// TIA Portal project "SimLogic" (V15)

(* hardware
DEVICE "S71500/ET200MP station_1"  S7-1500 station
   slot 0: "Rail_0"  Rack  6ES7 590-1***0-0AA0
   slot 1: "PLC_1"  CPU 1511-1 PN  6ES7 511-1AK00-0AB0  V1.8
      slot 3: "CPU display_1"  6ES7591-1AA00-0AA0
DEVICE "PC-System_1"  SIMATIC PC station
   slot 0: "SIMATIC PC station"  Rail  SIMATIC PC-Station  V1.0
      slot 125: "Stationmanager"  Station_Manager  V6.0.4
   slot 1: "HMI_RT_1"  WinCC RT Professional  6AV2 105-0xxxx-xxxx  15.0.0.0
   slot 2: "IE general_1"  IE General  IE_CP  V8.2.0
*)

// ===== PLC "PLC_1"  CPU 1511-1 PN =====

VAR_GLOBAL   // PLC tag table "Default tag table"
   "Brake_Out" AT %M0.0 : Bool;
   "Baffle_Out" AT %MW18 : Int;
   "RPM_In" AT %MW2 : Int;
   "OilTemp_In" AT %MW4 : Int;
   "Baffle_En" AT %M0.1 : Bool;
   "Current_In" AT %MW6 : Int;
   "OilPumpVFDsp_Out" AT %MW8 : Int;
   "OilPumpVFDen_Out" AT %M0.2 : Bool;
   "OilFlow_In" AT %MW10 : Int;
   "ProgLang" AT %MW12 : Int;
   "ONS1" AT %M0.3 : Bool;
   "PB_LAD" AT %M0.4 : Bool;
   "ONS" AT %M0.5 : Bool;
   "PB_FBD" AT %M0.6 : Bool;
   "PB_SCL" AT %M0.7 : Bool;
   "PB_STL" AT %M1.0 : Bool;
   "ONS2" AT %M1.1 : Bool;
   "ONS3" AT %M1.2 : Bool;
   "ONS4" AT %M1.3 : Bool;
   "AlarmHorn_Out" AT %M1.4 : Bool;
   "StationInterlock_Out" AT %M1.5 : Bool;
   "OilPumpVFDsp_Pct" AT %MW14 : Int;
   "Baffle_Pct" AT %MW16 : Int;
   "OilTemp" AT %MW20 : Int;
   "OilFlow" AT %MW22 : Int;
   "RPM" AT %MW24 : Int;
   "Current" AT %MW26 : Int;
   "OilPumpVFDOff_PB" AT %M1.6 : Bool;
   "OilPumpVFDHand_PB" AT %M1.7 : Bool;
   "OilPumpVFDAuto_PB" AT %M28.0 : Bool;
   "OilPumpVFD_HOA" AT %MW30 : Int;
   "Brake_HOA" AT %MW32 : Int;
   "BrakeOff_PB" AT %M28.1 : Bool;
   "BrakeHand_PB" AT %M28.2 : Bool;
   "BrakeAuto_PB" AT %M28.3 : Bool;
   "AlarmHorn_HOA" AT %MW34 : Int;
   "AlarmHornOff_PB" AT %M28.4 : Bool;
   "AlarmHornHand_PB" AT %M28.5 : Bool;
   "AlarmHornAuto_PB" AT %M28.6 : Bool;
   "StationIntOff_PB" AT %M28.7 : Bool;
   "StationIntHand_PB" AT %M29.0 : Bool;
   "StationIntAuto_PB" AT %M29.1 : Bool;
   "StationInt_HOA" AT %MW36 : Int;
   "StationInt" AT %M29.2 : Bool;
   "Brake_Ctrl" AT %M29.3 : Bool;
   "AlarmHorn_Ctrl" AT %M29.4 : Bool;
   "StationInt_Ctrl" AT %M29.5 : Bool;
   "OilPumpVFD_Ctrl" AT %M29.6 : Bool;
   "OilLowFlowDelay_SP" AT %MW38 : Int;
   "AlarmReset" AT %M29.7 : Bool;
   "AlarmSilence" AT %M40.0 : Bool;
   "OilLowFlowAlarm" AT %M40.1 : Bool;
   "OilLowFlowNotify" AT %M40.2 : Bool;
   "OilLowFlowAlarm_SP" AT %MW42 : Int;
   "OvercurrentDelay_SP" AT %MW44 : Int;
   "OvercurrentAlarm_SP" AT %MW46 : Int;
   "OvercurrentAlarm" AT %M40.3 : Bool;
   "OvercurrentNotify" AT %M40.4 : Bool;
   "HighOilTempDelay_SP" AT %MW48 : Int;
   "HighOilTempAlarm_SP" AT %MW50 : Int;
   "HighOilTempAlarm" AT %M40.5 : Bool;
   "HighOilTempNotify" AT %M40.6 : Bool;
   "RotorOverspeedDelay_SP" AT %MW52 : Int;
   "RotorOverspeedAlarm_SP" AT %MW54 : Int;
   "RotorOverspeedAlarm" AT %M40.7 : Bool;
   "RotorOverspeedNotify" AT %M41.0 : Bool;
   "OilHighFlowDelay_SP" AT %MW56 : Int;
   "OilHighFlowAlarm_SP" AT %MW58 : Int;
   "OilHighFlowAlarm" AT %M41.1 : Bool;
   "OilHighFlowNotify" AT %M41.2 : Bool;
   "BrakeFailureDelay_SP" AT %MW60 : Int;
   "BrakeFailureAlarm" AT %M41.3 : Bool;
   "BrakeFailureNotify" AT %M41.4 : Bool;
   "EStop" AT %M41.5 : Bool;
   "EStopAlarm" AT %M41.6 : Bool;
   "EStopNotify" AT %M41.7 : Bool;
   "AlarmReset_PB" AT %M62.0 : Bool;
   "AlarmSilence_PB" AT %M62.1 : Bool;
   "Baffle_HOA" AT %MW64 : Int;
   "Baffle_Ctrl" AT %M62.2 : Bool;
   "BaffleEn_Out" AT %M62.3 : Bool;
   "WarmupMode" AT %M62.4 : Bool;
   "WarmupRPM" AT %MW66 : Int;
   "BafflePID_SP" AT %MW68 : Int;
   "WarmupVFD_Pct" AT %MW70 : Int;
   "VFD_SP" AT %MW72 : Int;
   "WarmupOilTemp_SP" AT %MW74 : Int;
   "WarmupOilTempDelay_SP" AT %MW76 : Int;
   "WarmupTransition" AT %M62.5 : Bool;
   "BafflePID_In" AT %MW78 : Int;
   "StabilizeMode" AT %M62.6 : Bool;
   "StabilizekW_SP" AT %MW80 : Int;
   "StabilizeDelay_SP" AT %MW82 : Int;
   "StabilizeTransition" AT %M62.7 : Bool;
   "GenerationMode" AT %M63.0 : Bool;
   "SystemStart_PB" AT %M63.1 : Bool;
   "StartSequenceBit" AT %M63.2 : Bool;
   "SystemStop_PB" AT %M63.3 : Bool;
   "GenerationTransition" AT %M63.4 : Bool;
   "CooldownMode" AT %M63.5 : Bool;
   "CooldownRPM" AT %MW84 : Int;
   "CooldownDelay_SP" AT %MW86 : Int;
   "CooldownTransition" AT %M63.6 : Bool;
   "CooldownRPM_SP" AT %MW88 : Int;
   "CooldownOilTemp_SP" AT %MW90 : Int;
   "IdleMode" AT %M63.7 : Bool;
   "FaultMode" AT %M92.0 : Bool;
   "SequenceRunning" AT %M92.1 : Bool;
   "ONS5" AT %M92.2 : Bool;
   "ONS6" AT %M92.3 : Bool;
   "VFDOHFOverride_SP" AT %MW94 : Int;
   "ONS7" AT %M92.4 : Bool;
   "BaffleManual" AT %M92.5 : Bool;
   "BaffleAuto_PB" AT %M92.6 : Bool;
   "ONS8" AT %M92.7 : Bool;
   "BaffleHand_PB" AT %M93.0 : Bool;
   "BaffleOff_PB" AT %M93.1 : Bool;
   "ONS9" AT %M93.2 : Bool;
   "BaffleManual_SP" AT %MD96 : Real;
   "ONS10" AT %M93.3 : Bool;
   "ONS11" AT %M93.4 : Bool;
   "VFDHand_PB" AT %M93.5 : Bool;
   "VFD_HOA" AT %MW100 : Int;
   "VFDOff_PB" AT %M93.6 : Bool;
   "ONS16" AT %M93.7 : Bool;
   "ONS12" AT %M102.0 : Bool;
   "VFDAuto_PB" AT %M102.1 : Bool;
   "ONS13" AT %M102.2 : Bool;
   "VFDManual_SP" AT %MD104 : Real;
   "ONS14" AT %M102.3 : Bool;
   "ONS15" AT %M102.4 : Bool;
   "VFDManual" AT %M102.5 : Bool;
   "OilPumpVFD_On" AT %M102.6 : Bool;
   "BafflePID_On" AT %M102.7 : Bool;
   "FullAutoBit" AT %M103.0 : Bool;
   "HM_Minutes" AT %MW108 : Int;
   "HM_Hours" AT %MW110 : Int;
   "HM_Days" AT %MW112 : Int;
   "ResetHourmeter_PB" AT %M103.1 : Bool;
   "ModeInt" AT %MW114 : Int;
END_VAR

DATA_BLOCK "SimLogic_DB"   // DB1
{ S7_Optimized_Access := 'TRUE' }
VERSION : 0.1
// stored: InstanceOfName SimLogic
"SimLogic"
BEGIN
END_DATA_BLOCK

DATA_BLOCK "IO_LAD_DB"   // DB2
{ S7_Optimized_Access := 'TRUE' }
VERSION : 0.1
// stored: InstanceOfName IO_LAD
"IO_LAD"
BEGIN
END_DATA_BLOCK

DATA_BLOCK "IO_FBD_DB"   // DB4
{ S7_Optimized_Access := 'TRUE' }
VERSION : 0.1
// stored: InstanceOfName IO_FBD
"IO_FBD"
BEGIN
END_DATA_BLOCK

DATA_BLOCK "IO_SCL_DB"   // DB5
{ S7_Optimized_Access := 'TRUE' }
VERSION : 0.1
// stored: InstanceOfName IO_SCL
"IO_SCL"
BEGIN
END_DATA_BLOCK

DATA_BLOCK "IO_STL_DB"   // DB6
{ S7_Optimized_Access := 'TRUE' }
VERSION : 0.1
// stored: InstanceOfName IO_STL
"IO_STL"
BEGIN
END_DATA_BLOCK

DATA_BLOCK "HOA_LAD_DB"   // DB7
{ S7_Optimized_Access := 'TRUE' }
VERSION : 0.1
// stored: InstanceOfName HOA_LAD
"HOA_LAD"
BEGIN
END_DATA_BLOCK

DATA_BLOCK "HOA_FBD_DB"   // DB8
{ S7_Optimized_Access := 'TRUE' }
VERSION : 0.1
// stored: InstanceOfName HOA_FBD
"HOA_FBD"
BEGIN
END_DATA_BLOCK

DATA_BLOCK "HOA_SCL_DB"   // DB9
{ S7_Optimized_Access := 'TRUE' }
VERSION : 0.1
// stored: InstanceOfName HOA_SCL
"HOA_SCL"
BEGIN
END_DATA_BLOCK

DATA_BLOCK "HOA_STL_DB"   // DB10
{ S7_Optimized_Access := 'TRUE' }
VERSION : 0.1
// stored: InstanceOfName HOA_STL
"HOA_STL"
BEGIN
END_DATA_BLOCK

DATA_BLOCK "ALARMS_LAD_DB"   // DB11
{ S7_Optimized_Access := 'TRUE' }
VERSION : 0.1
// stored: InstanceOfName ALARMS_LAD
"ALARMS_LAD"
BEGIN
END_DATA_BLOCK

DATA_BLOCK "ALARMS_FBD_DB"   // DB12
{ S7_Optimized_Access := 'TRUE' }
VERSION : 0.1
// stored: InstanceOfName ALARMS_FBD
"ALARMS_FBD"
BEGIN
END_DATA_BLOCK

DATA_BLOCK "ALARMS_SCL_DB"   // DB13
{ S7_Optimized_Access := 'TRUE' }
VERSION : 0.1
// stored: InstanceOfName ALARMS_SCL
"ALARMS_SCL"
BEGIN
END_DATA_BLOCK

DATA_BLOCK "ALARMS_STL_DB"   // DB14
{ S7_Optimized_Access := 'TRUE' }
VERSION : 0.1
// stored: InstanceOfName ALARMS_STL
"ALARMS_STL"
BEGIN
END_DATA_BLOCK

DATA_BLOCK "MODES_LAD_DB"   // DB54
{ S7_Optimized_Access := 'TRUE' }
VERSION : 0.1
// stored: InstanceOfName MODES_LAD
"MODES_LAD"
BEGIN
END_DATA_BLOCK

DATA_BLOCK "MODES_FBD_DB"   // DB55
{ S7_Optimized_Access := 'TRUE' }
VERSION : 0.1
// stored: InstanceOfName MODES_FBD
"MODES_FBD"
BEGIN
END_DATA_BLOCK

DATA_BLOCK "MODES_SCL_DB"   // DB56
{ S7_Optimized_Access := 'TRUE' }
VERSION : 0.1
// stored: InstanceOfName MODES_SCL
"MODES_SCL"
BEGIN
END_DATA_BLOCK

DATA_BLOCK "MODES_STL_DB"   // DB57
{ S7_Optimized_Access := 'TRUE' }
VERSION : 0.1
// stored: InstanceOfName MODES_STL
"MODES_STL"
BEGIN
END_DATA_BLOCK

DATA_BLOCK "SEQUENCE_DB"   // DB58
{ S7_Optimized_Access := 'TRUE' }
VERSION : 0.1
// stored: InstanceOfName SEQUENCE
"SEQUENCE"
BEGIN
END_DATA_BLOCK

DATA_BLOCK "HOURMETER_LAD_DB"   // DB83
{ S7_Optimized_Access := 'TRUE' }
VERSION : 0.1
// stored: InstanceOfName HOURMETER_LAD
"HOURMETER_LAD"
BEGIN
END_DATA_BLOCK

DATA_BLOCK "HOURMETER_FBD_DB"   // DB84
{ S7_Optimized_Access := 'TRUE' }
VERSION : 0.1
// stored: InstanceOfName HOURMETER_FBD
"HOURMETER_FBD"
BEGIN
END_DATA_BLOCK

DATA_BLOCK "HOURMETER_SCL_DB"   // DB85
{ S7_Optimized_Access := 'TRUE' }
VERSION : 0.1
// stored: InstanceOfName HOURMETER_SCL
"HOURMETER_SCL"
BEGIN
END_DATA_BLOCK

DATA_BLOCK "HOURMETER_STL_DB"   // DB86
{ S7_Optimized_Access := 'TRUE' }
VERSION : 0.1
// stored: InstanceOfName HOURMETER_STL
"HOURMETER_STL"
BEGIN
END_DATA_BLOCK

// folder: System blocks/Program resources

DATA_BLOCK "IEC_Timer_0_DB_25"   // DB3
{ S7_Optimized_Access := 'TRUE' }
AUTHOR : Simatic
FAMILY : IEC
NAME : IEC_TMR
VERSION : 1.0
// stored: InstanceOfName IEC_TIMER
"IEC_TIMER"
BEGIN
END_DATA_BLOCK

DATA_BLOCK "IEC_Timer_0_DB_1"   // DB15
{ S7_Optimized_Access := 'TRUE' }
AUTHOR : Simatic
FAMILY : IEC
NAME : IEC_TMR
VERSION : 1.0
// stored: InstanceOfName IEC_TIMER
"IEC_TIMER"
BEGIN
END_DATA_BLOCK

DATA_BLOCK "IEC_Timer_0_DB_2"   // DB16
{ S7_Optimized_Access := 'TRUE' }
AUTHOR : Simatic
FAMILY : IEC
NAME : IEC_TMR
VERSION : 1.0
// stored: InstanceOfName IEC_TIMER
"IEC_TIMER"
BEGIN
END_DATA_BLOCK

DATA_BLOCK "IEC_Timer_0_DB"   // DB17
{ S7_Optimized_Access := 'TRUE' }
AUTHOR : Simatic
FAMILY : IEC
NAME : IEC_TMR
VERSION : 1.0
// stored: InstanceOfName IEC_TIMER
"IEC_TIMER"
BEGIN
END_DATA_BLOCK

DATA_BLOCK "IEC_Timer_0_DB_3"   // DB18
{ S7_Optimized_Access := 'TRUE' }
AUTHOR : Simatic
FAMILY : IEC
NAME : IEC_TMR
VERSION : 1.0
// stored: InstanceOfName IEC_TIMER
"IEC_TIMER"
BEGIN
END_DATA_BLOCK

DATA_BLOCK "IEC_Timer_0_DB_4"   // DB19
{ S7_Optimized_Access := 'TRUE' }
AUTHOR : Simatic
FAMILY : IEC
NAME : IEC_TMR
VERSION : 1.0
// stored: InstanceOfName IEC_TIMER
"IEC_TIMER"
BEGIN
END_DATA_BLOCK

DATA_BLOCK "IEC_Timer_0_DB_5"   // DB20
{ S7_Optimized_Access := 'TRUE' }
AUTHOR : Simatic
FAMILY : IEC
NAME : IEC_TMR
VERSION : 1.0
// stored: InstanceOfName IEC_TIMER
"IEC_TIMER"
BEGIN
END_DATA_BLOCK

DATA_BLOCK "IEC_Timer_0_DB_6"   // DB21
{ S7_Optimized_Access := 'TRUE' }
AUTHOR : Simatic
FAMILY : IEC
NAME : IEC_TMR
VERSION : 1.0
// stored: InstanceOfName IEC_TIMER
"IEC_TIMER"
BEGIN
END_DATA_BLOCK

DATA_BLOCK "IEC_Timer_0_DB_7"   // DB22
{ S7_Optimized_Access := 'TRUE' }
AUTHOR : Simatic
FAMILY : IEC
NAME : IEC_TMR
VERSION : 1.0
// stored: InstanceOfName IEC_TIMER
"IEC_TIMER"
BEGIN
END_DATA_BLOCK

DATA_BLOCK "IEC_Timer_0_DB_8"   // DB23
{ S7_Optimized_Access := 'TRUE' }
AUTHOR : Simatic
FAMILY : IEC
NAME : IEC_TMR
VERSION : 1.0
// stored: InstanceOfName IEC_TIMER
"IEC_TIMER"
BEGIN
END_DATA_BLOCK

DATA_BLOCK "IEC_Timer_0_DB_9"   // DB24
{ S7_Optimized_Access := 'TRUE' }
AUTHOR : Simatic
FAMILY : IEC
NAME : IEC_TMR
VERSION : 1.0
// stored: InstanceOfName IEC_TIMER
"IEC_TIMER"
BEGIN
END_DATA_BLOCK

DATA_BLOCK "IEC_Timer_0_DB_10"   // DB25
{ S7_Optimized_Access := 'TRUE' }
AUTHOR : Simatic
FAMILY : IEC
NAME : IEC_TMR
VERSION : 1.0
// stored: InstanceOfName IEC_TIMER
"IEC_TIMER"
BEGIN
END_DATA_BLOCK

DATA_BLOCK "IEC_Timer_0_DB_11"   // DB26
{ S7_Optimized_Access := 'TRUE' }
AUTHOR : Simatic
FAMILY : IEC
NAME : IEC_TMR
VERSION : 1.0
// stored: InstanceOfName IEC_TIMER
"IEC_TIMER"
BEGIN
END_DATA_BLOCK

DATA_BLOCK "IEC_Timer_0_DB_12"   // DB27
{ S7_Optimized_Access := 'TRUE' }
AUTHOR : Simatic
FAMILY : IEC
NAME : IEC_TMR
VERSION : 1.0
// stored: InstanceOfName IEC_TIMER
"IEC_TIMER"
BEGIN
END_DATA_BLOCK

DATA_BLOCK "IEC_Timer_0_DB_13"   // DB28
{ S7_Optimized_Access := 'TRUE' }
AUTHOR : Simatic
FAMILY : IEC
NAME : IEC_TMR
VERSION : 1.0
// stored: InstanceOfName IEC_TIMER
"IEC_TIMER"
BEGIN
END_DATA_BLOCK

DATA_BLOCK "IEC_Timer_0_DB_14"   // DB29
{ S7_Optimized_Access := 'TRUE' }
AUTHOR : Simatic
FAMILY : IEC
NAME : IEC_TMR
VERSION : 1.0
// stored: InstanceOfName IEC_TIMER
"IEC_TIMER"
BEGIN
END_DATA_BLOCK

DATA_BLOCK "IEC_Timer_0_DB_15"   // DB30
{ S7_Optimized_Access := 'TRUE' }
AUTHOR : Simatic
FAMILY : IEC
NAME : IEC_TMR
VERSION : 1.0
// stored: InstanceOfName IEC_TIMER
"IEC_TIMER"
BEGIN
END_DATA_BLOCK

DATA_BLOCK "IEC_Timer_0_DB_16"   // DB31
{ S7_Optimized_Access := 'TRUE' }
AUTHOR : Simatic
FAMILY : IEC
NAME : IEC_TMR
VERSION : 1.0
// stored: InstanceOfName IEC_TIMER
"IEC_TIMER"
BEGIN
END_DATA_BLOCK

DATA_BLOCK "IEC_Timer_0_DB_17"   // DB32
{ S7_Optimized_Access := 'TRUE' }
AUTHOR : Simatic
FAMILY : IEC
NAME : IEC_TMR
VERSION : 1.0
// stored: InstanceOfName IEC_TIMER
"IEC_TIMER"
BEGIN
END_DATA_BLOCK

DATA_BLOCK "IEC_Timer_0_DB_18"   // DB33
{ S7_Optimized_Access := 'TRUE' }
AUTHOR : Simatic
FAMILY : IEC
NAME : IEC_TMR
VERSION : 1.0
// stored: InstanceOfName IEC_TIMER
"IEC_TIMER"
BEGIN
END_DATA_BLOCK

DATA_BLOCK "IEC_Timer_0_DB_19"   // DB34
{ S7_Optimized_Access := 'TRUE' }
AUTHOR : Simatic
FAMILY : IEC
NAME : IEC_TMR
VERSION : 1.0
// stored: InstanceOfName IEC_TIMER
"IEC_TIMER"
BEGIN
END_DATA_BLOCK

DATA_BLOCK "IEC_Timer_0_DB_20"   // DB35
{ S7_Optimized_Access := 'TRUE' }
AUTHOR : Simatic
FAMILY : IEC
NAME : IEC_TMR
VERSION : 1.0
// stored: InstanceOfName IEC_TIMER
"IEC_TIMER"
BEGIN
END_DATA_BLOCK

DATA_BLOCK "IEC_Timer_0_DB_21"   // DB36
{ S7_Optimized_Access := 'TRUE' }
AUTHOR : Simatic
FAMILY : IEC
NAME : IEC_TMR
VERSION : 1.0
// stored: InstanceOfName IEC_TIMER
"IEC_TIMER"
BEGIN
END_DATA_BLOCK

DATA_BLOCK "IEC_Timer_0_DB_22"   // DB37
{ S7_Optimized_Access := 'TRUE' }
AUTHOR : Simatic
FAMILY : IEC
NAME : IEC_TMR
VERSION : 1.0
// stored: InstanceOfName IEC_TIMER
"IEC_TIMER"
BEGIN
END_DATA_BLOCK

DATA_BLOCK "IEC_Timer_0_DB_23"   // DB38
{ S7_Optimized_Access := 'TRUE' }
AUTHOR : Simatic
FAMILY : IEC
NAME : IEC_TMR
VERSION : 1.0
// stored: InstanceOfName IEC_TIMER
"IEC_TIMER"
BEGIN
END_DATA_BLOCK

DATA_BLOCK "IEC_Timer_0_DB_24"   // DB39
{ S7_Optimized_Access := 'TRUE' }
AUTHOR : Simatic
FAMILY : IEC
NAME : IEC_TMR
VERSION : 1.0
// stored: InstanceOfName IEC_TIMER
"IEC_TIMER"
BEGIN
END_DATA_BLOCK

DATA_BLOCK "IEC_Timer_0_DB_26"   // DB40
{ S7_Optimized_Access := 'TRUE' }
AUTHOR : Simatic
FAMILY : IEC
NAME : IEC_TMR
VERSION : 1.0
// stored: InstanceOfName IEC_TIMER
"IEC_TIMER"
BEGIN
END_DATA_BLOCK

DATA_BLOCK "IEC_Timer_0_DB_27"   // DB41
{ S7_Optimized_Access := 'TRUE' }
AUTHOR : Simatic
FAMILY : IEC
NAME : IEC_TMR
VERSION : 1.0
// stored: InstanceOfName IEC_TIMER
"IEC_TIMER"
BEGIN
END_DATA_BLOCK

DATA_BLOCK "IEC_Timer_1_DB"   // DB43
{ S7_Optimized_Access := 'TRUE' }
AUTHOR : Simatic
FAMILY : IEC
NAME : IEC_TMR
VERSION : 1.0
// stored: InstanceOfName IEC_TIMER
"IEC_TIMER"
BEGIN
END_DATA_BLOCK

DATA_BLOCK "IEC_Timer_0_DB_28"   // DB44
{ S7_Optimized_Access := 'TRUE' }
AUTHOR : Simatic
FAMILY : IEC
NAME : IEC_TMR
VERSION : 1.0
// stored: InstanceOfName IEC_TIMER
"IEC_TIMER"
BEGIN
END_DATA_BLOCK

DATA_BLOCK "IEC_Timer_0_DB_29"   // DB45
{ S7_Optimized_Access := 'TRUE' }
AUTHOR : Simatic
FAMILY : IEC
NAME : IEC_TMR
VERSION : 1.0
// stored: InstanceOfName IEC_TIMER
"IEC_TIMER"
BEGIN
END_DATA_BLOCK

DATA_BLOCK "IEC_Timer_0_DB_30"   // DB46
{ S7_Optimized_Access := 'TRUE' }
AUTHOR : Simatic
FAMILY : IEC
NAME : IEC_TMR
VERSION : 1.0
// stored: InstanceOfName IEC_TIMER
"IEC_TIMER"
BEGIN
END_DATA_BLOCK

DATA_BLOCK "IEC_Timer_0_DB_31"   // DB47
{ S7_Optimized_Access := 'TRUE' }
AUTHOR : Simatic
FAMILY : IEC
NAME : IEC_TMR
VERSION : 1.0
// stored: InstanceOfName IEC_TIMER
"IEC_TIMER"
BEGIN
END_DATA_BLOCK

DATA_BLOCK "IEC_Timer_0_DB_32"   // DB48
{ S7_Optimized_Access := 'TRUE' }
AUTHOR : Simatic
FAMILY : IEC
NAME : IEC_TMR
VERSION : 1.0
// stored: InstanceOfName IEC_TIMER
"IEC_TIMER"
BEGIN
END_DATA_BLOCK

DATA_BLOCK "IEC_Timer_0_DB_33"   // DB49
{ S7_Optimized_Access := 'TRUE' }
AUTHOR : Simatic
FAMILY : IEC
NAME : IEC_TMR
VERSION : 1.0
// stored: InstanceOfName IEC_TIMER
"IEC_TIMER"
BEGIN
END_DATA_BLOCK

DATA_BLOCK "IEC_Timer_0_DB_34"   // DB50
{ S7_Optimized_Access := 'TRUE' }
AUTHOR : Simatic
FAMILY : IEC
NAME : IEC_TMR
VERSION : 1.0
// stored: InstanceOfName IEC_TIMER
"IEC_TIMER"
BEGIN
END_DATA_BLOCK

DATA_BLOCK "IEC_Timer_0_DB_35"   // DB51
{ S7_Optimized_Access := 'TRUE' }
AUTHOR : Simatic
FAMILY : IEC
NAME : IEC_TMR
VERSION : 1.0
// stored: InstanceOfName IEC_TIMER
"IEC_TIMER"
BEGIN
END_DATA_BLOCK

DATA_BLOCK "IEC_Timer_0_DB_36"   // DB52
{ S7_Optimized_Access := 'TRUE' }
AUTHOR : Simatic
FAMILY : IEC
NAME : IEC_TMR
VERSION : 1.0
// stored: InstanceOfName IEC_TIMER
"IEC_TIMER"
BEGIN
END_DATA_BLOCK

DATA_BLOCK "IEC_Timer_0_DB_37"   // DB53
{ S7_Optimized_Access := 'TRUE' }
AUTHOR : Simatic
FAMILY : IEC
NAME : IEC_TMR
VERSION : 1.0
// stored: InstanceOfName IEC_TIMER
"IEC_TIMER"
BEGIN
END_DATA_BLOCK

DATA_BLOCK "IEC_Timer_0_DB_38"   // DB62
{ S7_Optimized_Access := 'TRUE' }
AUTHOR : Simatic
FAMILY : IEC
NAME : IEC_TMR
VERSION : 1.0
// stored: InstanceOfName IEC_TIMER
"IEC_TIMER"
BEGIN
END_DATA_BLOCK

DATA_BLOCK "IEC_Counter_0_DB"   // DB63
{ S7_Optimized_Access := 'TRUE' }
AUTHOR : Simatic
FAMILY : IEC
NAME : CNTR
VERSION : 1.0
// stored: InstanceOfName IEC_COUNTER
"IEC_COUNTER"
BEGIN
END_DATA_BLOCK

DATA_BLOCK "IEC_Counter_0_DB_1"   // DB64
{ S7_Optimized_Access := 'TRUE' }
AUTHOR : Simatic
FAMILY : IEC
NAME : CNTR
VERSION : 1.0
// stored: InstanceOfName IEC_COUNTER
"IEC_COUNTER"
BEGIN
END_DATA_BLOCK

DATA_BLOCK "IEC_Counter_0_DB_2"   // DB65
{ S7_Optimized_Access := 'TRUE' }
AUTHOR : Simatic
FAMILY : IEC
NAME : CNTR
VERSION : 1.0
// stored: InstanceOfName IEC_COUNTER
"IEC_COUNTER"
BEGIN
END_DATA_BLOCK

DATA_BLOCK "IEC_Timer_0_DB_39"   // DB66
{ S7_Optimized_Access := 'TRUE' }
AUTHOR : Simatic
FAMILY : IEC
NAME : IEC_TMR
VERSION : 1.0
// stored: InstanceOfName IEC_TIMER
"IEC_TIMER"
BEGIN
END_DATA_BLOCK

DATA_BLOCK "IEC_Timer_0_DB_40"   // DB67
{ S7_Optimized_Access := 'TRUE' }
AUTHOR : Simatic
FAMILY : IEC
NAME : IEC_TMR
VERSION : 1.0
// stored: InstanceOfName IEC_TIMER
"IEC_TIMER"
BEGIN
END_DATA_BLOCK

DATA_BLOCK "IEC_Timer_0_DB_41"   // DB68
{ S7_Optimized_Access := 'TRUE' }
AUTHOR : Simatic
FAMILY : IEC
NAME : IEC_TMR
VERSION : 1.0
// stored: InstanceOfName IEC_TIMER
"IEC_TIMER"
BEGIN
END_DATA_BLOCK

DATA_BLOCK "IEC_Counter_0_DB_3"   // DB69
{ S7_Optimized_Access := 'TRUE' }
AUTHOR : Simatic
FAMILY : IEC
NAME : CNTR
VERSION : 1.0
// stored: InstanceOfName IEC_COUNTER
"IEC_COUNTER"
BEGIN
END_DATA_BLOCK

DATA_BLOCK "IEC_Counter_0_DB_4"   // DB70
{ S7_Optimized_Access := 'TRUE' }
AUTHOR : Simatic
FAMILY : IEC
NAME : CNTR
VERSION : 1.0
// stored: InstanceOfName IEC_COUNTER
"IEC_COUNTER"
BEGIN
END_DATA_BLOCK

DATA_BLOCK "IEC_Timer_0_DB_42"   // DB71
{ S7_Optimized_Access := 'TRUE' }
AUTHOR : Simatic
FAMILY : IEC
NAME : IEC_TMR
VERSION : 1.0
// stored: InstanceOfName IEC_TIMER
"IEC_TIMER"
BEGIN
END_DATA_BLOCK

DATA_BLOCK "IEC_Counter_0_DB_5"   // DB72
{ S7_Optimized_Access := 'TRUE' }
AUTHOR : Simatic
FAMILY : IEC
NAME : CNTR
VERSION : 1.0
// stored: InstanceOfName IEC_COUNTER
"IEC_COUNTER"
BEGIN
END_DATA_BLOCK

DATA_BLOCK "IEC_Timer_0_DB_43"   // DB73
{ S7_Optimized_Access := 'TRUE' }
AUTHOR : Simatic
FAMILY : IEC
NAME : IEC_TMR
VERSION : 1.0
// stored: InstanceOfName IEC_TIMER
"IEC_TIMER"
BEGIN
END_DATA_BLOCK

DATA_BLOCK "IEC_Counter_0_DB_6"   // DB74
{ S7_Optimized_Access := 'TRUE' }
AUTHOR : Simatic
FAMILY : IEC
NAME : CNTR
VERSION : 1.0
// stored: InstanceOfName IEC_COUNTER
"IEC_COUNTER"
BEGIN
END_DATA_BLOCK

DATA_BLOCK "IEC_Counter_0_DB_7"   // DB75
{ S7_Optimized_Access := 'TRUE' }
AUTHOR : Simatic
FAMILY : IEC
NAME : CNTR
VERSION : 1.0
// stored: InstanceOfName IEC_COUNTER
"IEC_COUNTER"
BEGIN
END_DATA_BLOCK

DATA_BLOCK "IEC_Counter_0_DB_8"   // DB76
{ S7_Optimized_Access := 'TRUE' }
AUTHOR : Simatic
FAMILY : IEC
NAME : CNTR
VERSION : 1.0
// stored: InstanceOfName IEC_COUNTER
"IEC_COUNTER"
BEGIN
END_DATA_BLOCK

DATA_BLOCK "IEC_Timer_0_DB_44"   // DB77
{ S7_Optimized_Access := 'TRUE' }
AUTHOR : Simatic
FAMILY : IEC
NAME : IEC_TMR
VERSION : 1.0
// stored: InstanceOfName IEC_TIMER
"IEC_TIMER"
BEGIN
END_DATA_BLOCK

DATA_BLOCK "IEC_Timer_0_DB_45"   // DB78
{ S7_Optimized_Access := 'TRUE' }
AUTHOR : Simatic
FAMILY : IEC
NAME : IEC_TMR
VERSION : 1.0
// stored: InstanceOfName IEC_TIMER
"IEC_TIMER"
BEGIN
END_DATA_BLOCK

DATA_BLOCK "IEC_Counter_0_DB_9"   // DB79
{ S7_Optimized_Access := 'TRUE' }
AUTHOR : Simatic
FAMILY : IEC
NAME : CNTR
VERSION : 1.0
// stored: InstanceOfName IEC_COUNTER
"IEC_COUNTER"
BEGIN
END_DATA_BLOCK

DATA_BLOCK "IEC_Counter_0_DB_10"   // DB80
{ S7_Optimized_Access := 'TRUE' }
AUTHOR : Simatic
FAMILY : IEC
NAME : CNTR
VERSION : 1.0
// stored: InstanceOfName IEC_COUNTER
"IEC_COUNTER"
BEGIN
END_DATA_BLOCK

DATA_BLOCK "IEC_Counter_0_DB_11"   // DB81
{ S7_Optimized_Access := 'TRUE' }
AUTHOR : Simatic
FAMILY : IEC
NAME : CNTR
VERSION : 1.0
// stored: InstanceOfName IEC_COUNTER
"IEC_COUNTER"
BEGIN
END_DATA_BLOCK

DATA_BLOCK "IEC_Timer_0_DB_46"   // DB82
{ S7_Optimized_Access := 'TRUE' }
AUTHOR : Simatic
FAMILY : IEC
NAME : IEC_TMR
VERSION : 1.0
// stored: InstanceOfName IEC_TIMER
"IEC_TIMER"
BEGIN
END_DATA_BLOCK

// folder: (top level)

FUNCTION_BLOCK "SimLogic"   // FB1, FBD
{ S7_Optimized_Access := 'TRUE' }
VERSION : 0.1
   VAR
      "TO" : Bool;
      rpmv : Int;
      addrpmv : Bool;
      otsp : Int;
      ott : Int;
      TO1 : Bool;
      TO2 : Bool;
      be2 : Int;
      be3 : Int;
      be1 : Int;
      TO3 : Bool;
   END_VAR
   VAR_TEMP
      bf : Int;
      rpmvt : Int;
      bfr : Real;
   END_VAR
BEGIN

REGION Network 1
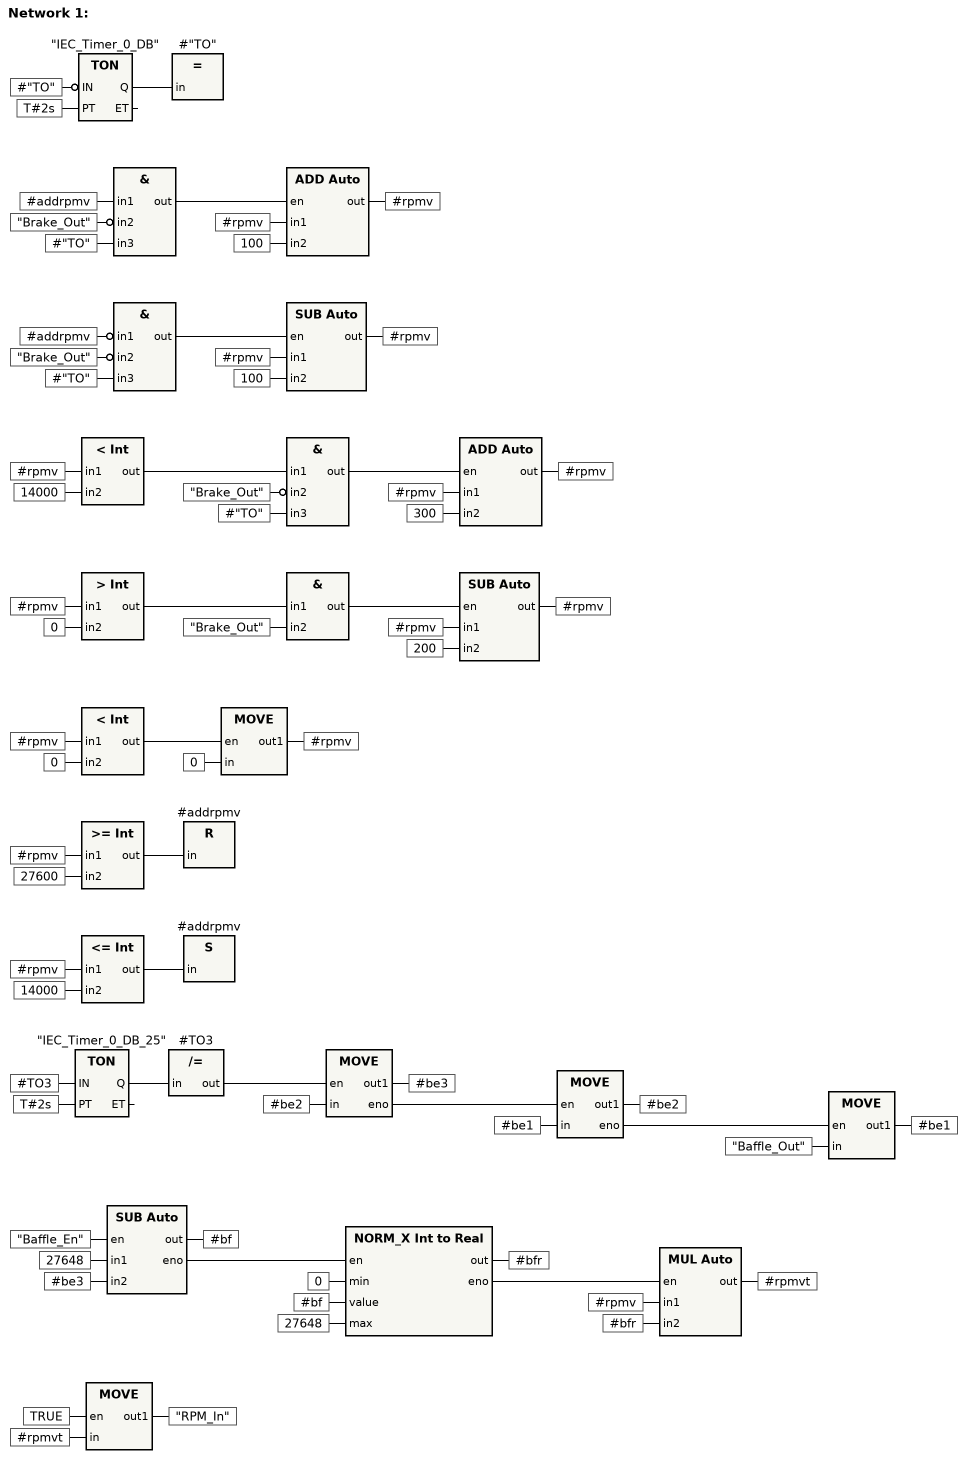
   "IEC_Timer_0_DB".TON(IN := NOT #"TO", PT := T#2s);
   #"TO" := "IEC_Timer_0_DB".Q;
   IF #addrpmv AND NOT "Brake_Out" AND #"TO" THEN #rpmv := #rpmv + 100; END_IF;
   IF NOT #addrpmv AND NOT "Brake_Out" AND #"TO" THEN #rpmv := #rpmv - 100; END_IF;
   IF (#rpmv < 14000) AND NOT "Brake_Out" AND #"TO" THEN #rpmv := #rpmv + 300; END_IF;
   IF (#rpmv > 0) AND "Brake_Out" THEN #rpmv := #rpmv - 200; END_IF;
   IF #rpmv < 0 THEN #rpmv := 0; END_IF;
   IF #rpmv >= 27600 THEN #addrpmv := FALSE; END_IF;
   IF #rpmv <= 14000 THEN #addrpmv := TRUE; END_IF;
   "IEC_Timer_0_DB_25".TON(IN := #TO3, PT := T#2s);
   #TO3 := NOT "IEC_Timer_0_DB_25".Q;
   IF "IEC_Timer_0_DB_25".Q THEN
       #be3 := #be2;
       #be2 := #be1;
       #be1 := "Baffle_Out";
   END_IF;
   IF "Baffle_En" THEN
       #bf := 27648 - #be3;
       #bfr := NORM_X(MIN := 0, VALUE := #bf, MAX := 27648);
       #rpmvt := #rpmv * #bfr;
   END_IF;
   IF TRUE THEN "RPM_In" := #rpmvt; END_IF;
END_REGION

REGION Network 2
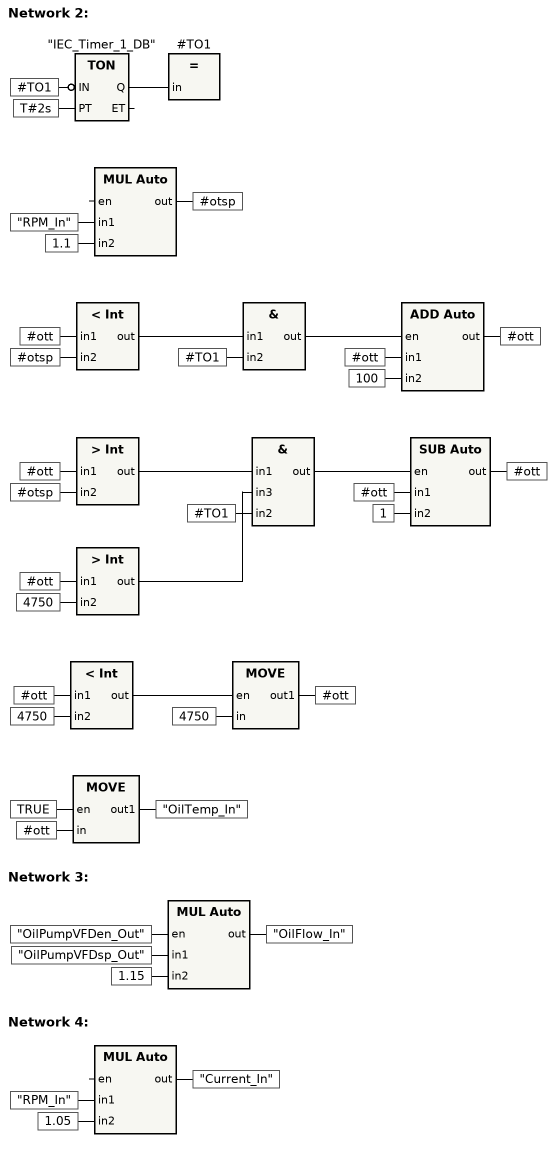
   "IEC_Timer_1_DB".TON(IN := NOT #TO1, PT := T#2s);
   #TO1 := "IEC_Timer_1_DB".Q;
   #otsp := "RPM_In" * 1.1;
   IF (#ott < #otsp) AND #TO1 THEN #ott := #ott + 100; END_IF;
   IF (#ott > #otsp) AND (#ott > 4750) AND #TO1 THEN #ott := #ott - 1; END_IF;
   IF #ott < 4750 THEN #ott := 4750; END_IF;
   IF TRUE THEN "OilTemp_In" := #ott; END_IF;
END_REGION

REGION Network 3
   IF "OilPumpVFDen_Out" THEN "OilFlow_In" := "OilPumpVFDsp_Out" * 1.15; END_IF;
END_REGION

REGION Network 4
   "Current_In" := "RPM_In" * 1.05;
END_REGION
END_FUNCTION_BLOCK

FUNCTION_BLOCK "IO_LAD"   // FB2, LAD
{ S7_Optimized_Access := 'TRUE' }
VERSION : 0.1
BEGIN

REGION Network 1
   // Digital Outputs
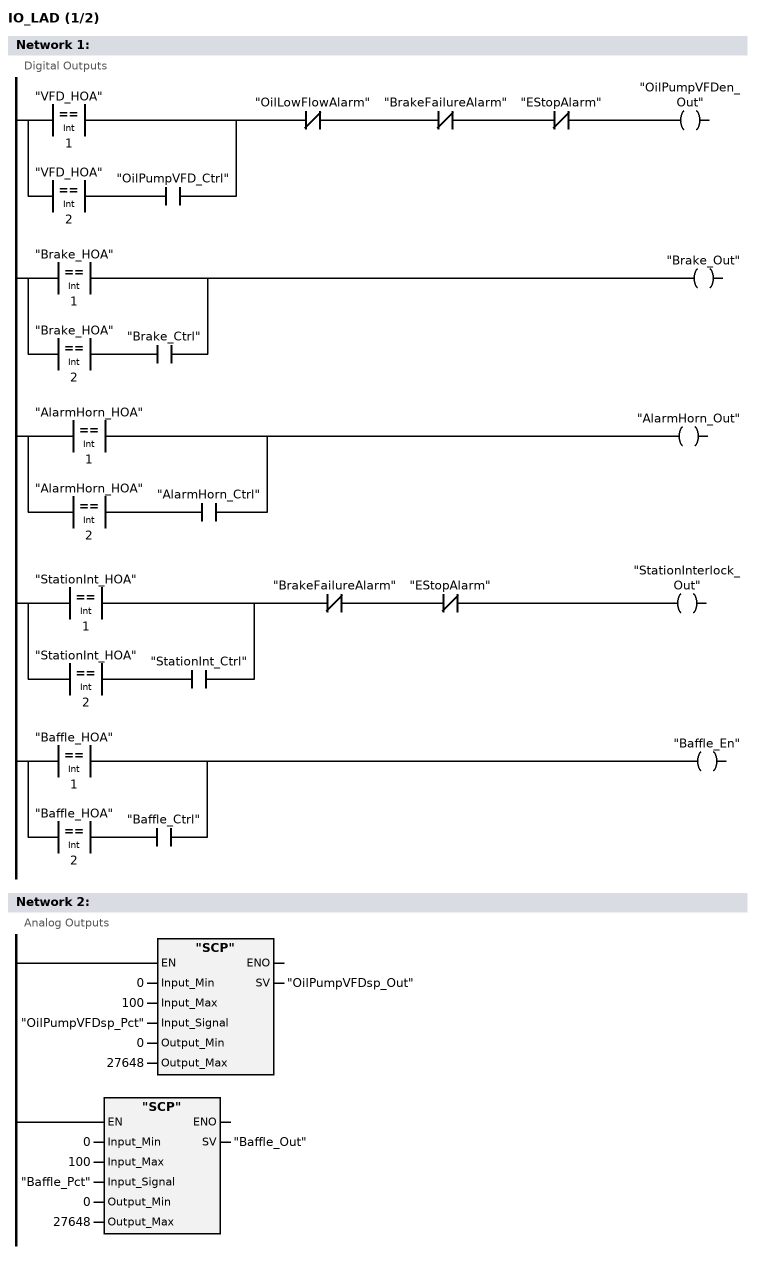
   RUNG wire#powerrail
      { S7_Templates := "SrcType := Int" } EQ_Contact(in1 := "VFD_HOA", in2 := 1)
      wire#w1
      I_Contact( "OilLowFlowAlarm" )
      I_Contact( "BrakeFailureAlarm" )
      I_Contact( "EStopAlarm" )
      Coil( "OilPumpVFDen_Out" )
   END_RUNG
   RUNG wire#powerrail
      { S7_Templates := "SrcType := Int" } EQ_Contact(in1 := "VFD_HOA", in2 := 2)
      Contact( "OilPumpVFD_Ctrl" )
   END_RUNG wire#w1
   RUNG wire#powerrail
      { S7_Templates := "SrcType := Int" } EQ_Contact(in1 := "Brake_HOA", in2 := 1)
      wire#w2
      Coil( "Brake_Out" )
   END_RUNG
   RUNG wire#powerrail
      { S7_Templates := "SrcType := Int" } EQ_Contact(in1 := "Brake_HOA", in2 := 2)
      Contact( "Brake_Ctrl" )
   END_RUNG wire#w2
   RUNG wire#powerrail
      { S7_Templates := "SrcType := Int" } EQ_Contact(in1 := "AlarmHorn_HOA", in2 := 1)
      wire#w3
      Coil( "AlarmHorn_Out" )
   END_RUNG
   RUNG wire#powerrail
      { S7_Templates := "SrcType := Int" } EQ_Contact(in1 := "AlarmHorn_HOA", in2 := 2)
      Contact( "AlarmHorn_Ctrl" )
   END_RUNG wire#w3
   RUNG wire#powerrail
      { S7_Templates := "SrcType := Int" } EQ_Contact(in1 := "StationInt_HOA", in2 := 1)
      wire#w4
      I_Contact( "BrakeFailureAlarm" )
      I_Contact( "EStopAlarm" )
      Coil( "StationInterlock_Out" )
   END_RUNG
   RUNG wire#powerrail
      { S7_Templates := "SrcType := Int" } EQ_Contact(in1 := "StationInt_HOA", in2 := 2)
      Contact( "StationInt_Ctrl" )
   END_RUNG wire#w4
   RUNG wire#powerrail
      { S7_Templates := "SrcType := Int" } EQ_Contact(in1 := "Baffle_HOA", in2 := 1)
      wire#w5
      Coil( "Baffle_En" )
   END_RUNG
   RUNG wire#powerrail
      { S7_Templates := "SrcType := Int" } EQ_Contact(in1 := "Baffle_HOA", in2 := 2)
      Contact( "Baffle_Ctrl" )
   END_RUNG wire#w5
   // the same network as SCL:
   "OilPumpVFDen_Out" := (("VFD_HOA" = 1) OR (("VFD_HOA" = 2) AND "OilPumpVFD_Ctrl")) AND NOT "OilLowFlowAlarm" AND NOT "BrakeFailureAlarm" AND NOT "EStopAlarm";
   "Brake_Out" := ("Brake_HOA" = 1) OR (("Brake_HOA" = 2) AND "Brake_Ctrl");
   "AlarmHorn_Out" := ("AlarmHorn_HOA" = 1) OR (("AlarmHorn_HOA" = 2) AND "AlarmHorn_Ctrl");
   "StationInterlock_Out" := (("StationInt_HOA" = 1) OR (("StationInt_HOA" = 2) AND "StationInt_Ctrl")) AND NOT "BrakeFailureAlarm" AND NOT "EStopAlarm";
   "Baffle_En" := ("Baffle_HOA" = 1) OR (("Baffle_HOA" = 2) AND "Baffle_Ctrl");
END_REGION

REGION Network 2
   // Analog Outputs
   RUNG wire#powerrail
      "SCP"(Input_Min := 0, Input_Max := 100, Input_Signal := "OilPumpVFDsp_Pct", Output_Min := 0, Output_Max := 27648, SV => "OilPumpVFDsp_Out")
   END_RUNG
   RUNG wire#powerrail
      "SCP"(Input_Min := 0, Input_Max := 100, Input_Signal := "Baffle_Pct", Output_Min := 0, Output_Max := 27648, SV => "Baffle_Out")
   END_RUNG
   // the same network as SCL:
   "SCP"(Input_Min := 0,
         Input_Max := 100,
         Input_Signal := "OilPumpVFDsp_Pct",
         Output_Min := 0,
         Output_Max := 27648,
         SV => "OilPumpVFDsp_Out");
   "SCP"(Input_Min := 0,
         Input_Max := 100,
         Input_Signal := "Baffle_Pct",
         Output_Min := 0,
         Output_Max := 27648,
         SV => "Baffle_Out");
END_REGION

REGION Network 3
   // Analog Inputs
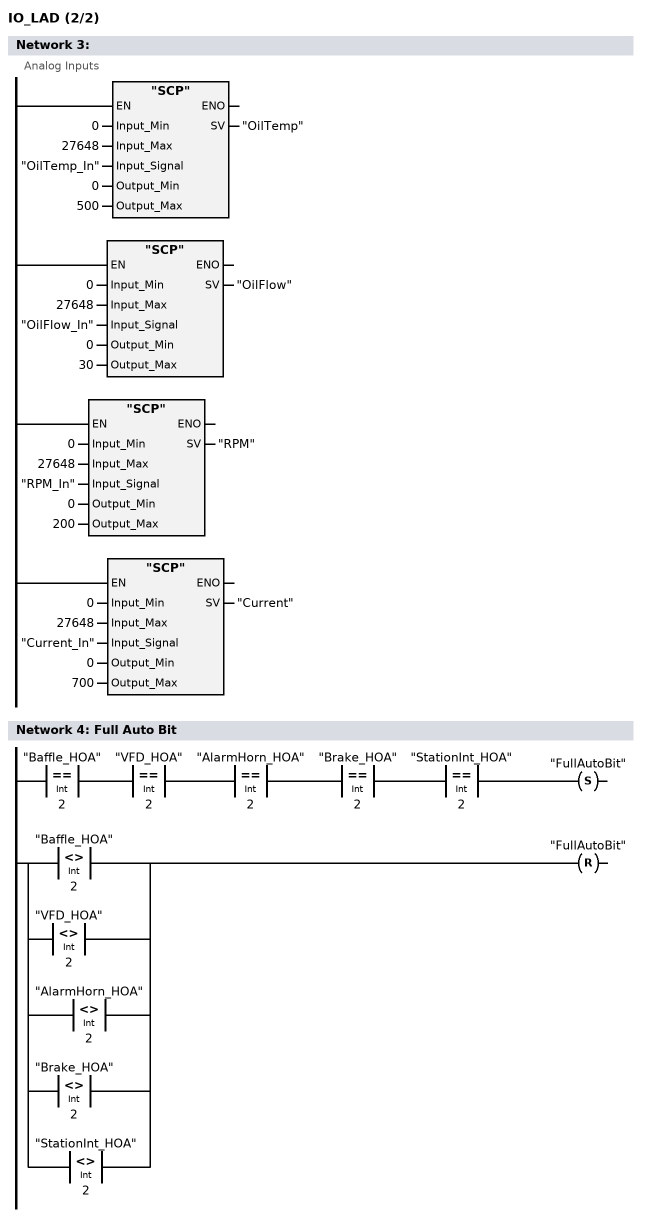
   RUNG wire#powerrail
      "SCP"(Input_Min := 0, Input_Max := 27648, Input_Signal := "OilTemp_In", Output_Min := 0, Output_Max := 500, SV => "OilTemp")
   END_RUNG
   RUNG wire#powerrail
      "SCP"(Input_Min := 0, Input_Max := 27648, Input_Signal := "OilFlow_In", Output_Min := 0, Output_Max := 30, SV => "OilFlow")
   END_RUNG
   RUNG wire#powerrail
      "SCP"(Input_Min := 0, Input_Max := 27648, Input_Signal := "RPM_In", Output_Min := 0, Output_Max := 200, SV => "RPM")
   END_RUNG
   RUNG wire#powerrail
      "SCP"(Input_Min := 0, Input_Max := 27648, Input_Signal := "Current_In", Output_Min := 0, Output_Max := 700, SV => "Current")
   END_RUNG
   // the same network as SCL:
   "SCP"(Input_Min := 0,
         Input_Max := 27648,
         Input_Signal := "OilTemp_In",
         Output_Min := 0,
         Output_Max := 500,
         SV => "OilTemp");
   "SCP"(Input_Min := 0,
         Input_Max := 27648,
         Input_Signal := "OilFlow_In",
         Output_Min := 0,
         Output_Max := 30,
         SV => "OilFlow");
   "SCP"(Input_Min := 0,
         Input_Max := 27648,
         Input_Signal := "RPM_In",
         Output_Min := 0,
         Output_Max := 200,
         SV => "RPM");
   "SCP"(Input_Min := 0,
         Input_Max := 27648,
         Input_Signal := "Current_In",
         Output_Min := 0,
         Output_Max := 700,
         SV => "Current");
END_REGION

REGION Network 4: Full Auto Bit
   RUNG wire#powerrail
      { S7_Templates := "SrcType := Int" } EQ_Contact(in1 := "Baffle_HOA", in2 := 2)
      { S7_Templates := "SrcType := Int" } EQ_Contact(in1 := "VFD_HOA", in2 := 2)
      { S7_Templates := "SrcType := Int" } EQ_Contact(in1 := "AlarmHorn_HOA", in2 := 2)
      { S7_Templates := "SrcType := Int" } EQ_Contact(in1 := "Brake_HOA", in2 := 2)
      { S7_Templates := "SrcType := Int" } EQ_Contact(in1 := "StationInt_HOA", in2 := 2)
      S_Coil( "FullAutoBit" )
   END_RUNG
   RUNG wire#powerrail
      { S7_Templates := "SrcType := Int" } NE_Contact(in1 := "Baffle_HOA", in2 := 2)
      wire#w1
      R_Coil( "FullAutoBit" )
   END_RUNG
   RUNG wire#powerrail
      { S7_Templates := "SrcType := Int" } NE_Contact(in1 := "VFD_HOA", in2 := 2)
   END_RUNG wire#w1
   RUNG wire#powerrail
      { S7_Templates := "SrcType := Int" } NE_Contact(in1 := "AlarmHorn_HOA", in2 := 2)
   END_RUNG wire#w1
   RUNG wire#powerrail
      { S7_Templates := "SrcType := Int" } NE_Contact(in1 := "Brake_HOA", in2 := 2)
   END_RUNG wire#w1
   RUNG wire#powerrail
      { S7_Templates := "SrcType := Int" } NE_Contact(in1 := "StationInt_HOA", in2 := 2)
   END_RUNG wire#w1
   // the same network as SCL:
   IF ("Baffle_HOA" = 2) AND ("VFD_HOA" = 2) AND ("AlarmHorn_HOA" = 2) AND ("Brake_HOA" = 2) AND ("StationInt_HOA" = 2) THEN
       "FullAutoBit" := TRUE;
   END_IF;
   IF ("Baffle_HOA" <> 2) OR ("VFD_HOA" <> 2) OR ("AlarmHorn_HOA" <> 2) OR ("Brake_HOA" <> 2) OR ("StationInt_HOA" <> 2) THEN
       "FullAutoBit" := FALSE;
   END_IF;
END_REGION
END_FUNCTION_BLOCK

FUNCTION_BLOCK "IO_FBD"   // FB3, FBD
{ S7_Optimized_Access := 'TRUE' }
VERSION : 0.1
BEGIN

REGION Network 1
   // Digital Outputs
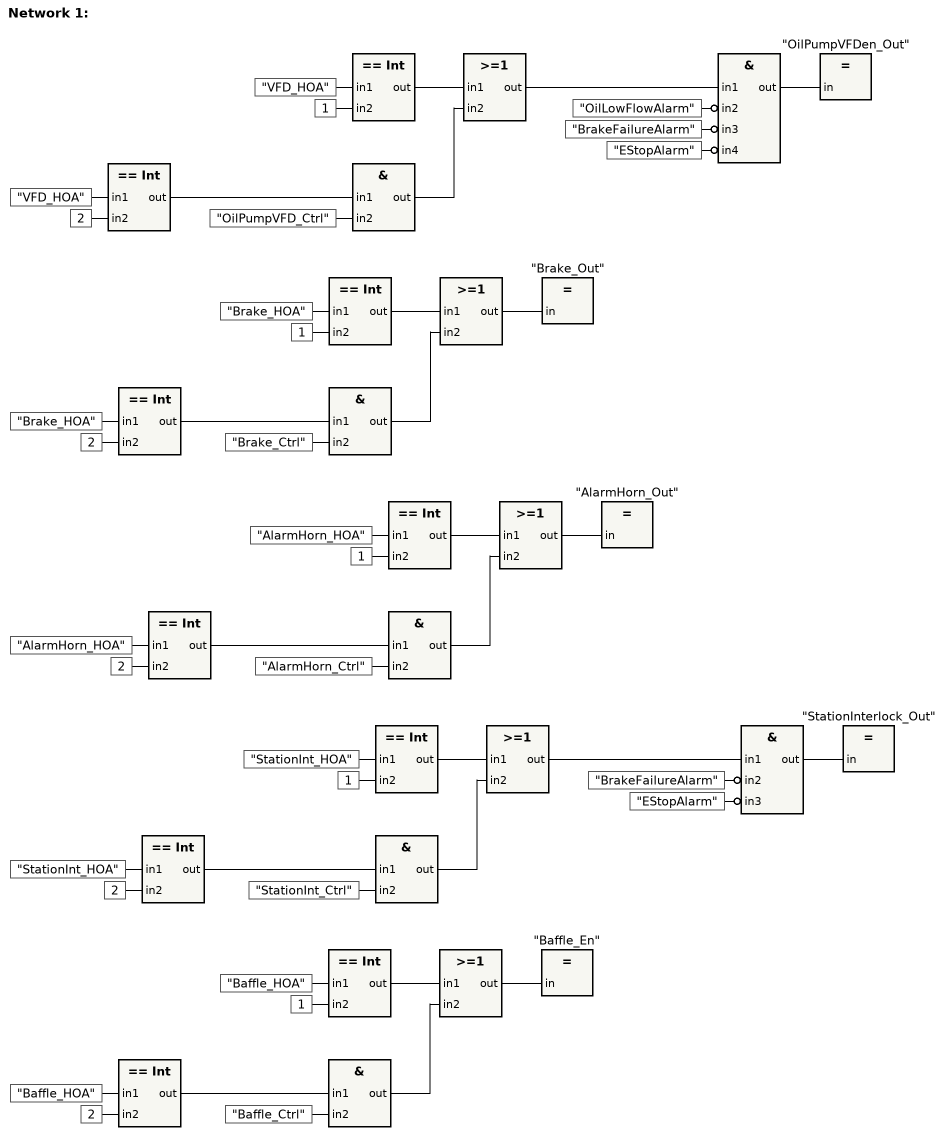
   "OilPumpVFDen_Out" := (("VFD_HOA" = 1) OR (("VFD_HOA" = 2) AND "OilPumpVFD_Ctrl")) AND NOT "OilLowFlowAlarm" AND NOT "BrakeFailureAlarm" AND NOT "EStopAlarm";
   "Brake_Out" := ("Brake_HOA" = 1) OR (("Brake_HOA" = 2) AND "Brake_Ctrl");
   "AlarmHorn_Out" := ("AlarmHorn_HOA" = 1) OR (("AlarmHorn_HOA" = 2) AND "AlarmHorn_Ctrl");
   "StationInterlock_Out" := (("StationInt_HOA" = 1) OR (("StationInt_HOA" = 2) AND "StationInt_Ctrl")) AND NOT "BrakeFailureAlarm" AND NOT "EStopAlarm";
   "Baffle_En" := ("Baffle_HOA" = 1) OR (("Baffle_HOA" = 2) AND "Baffle_Ctrl");
END_REGION

REGION Network 2
   // Analog Outputs
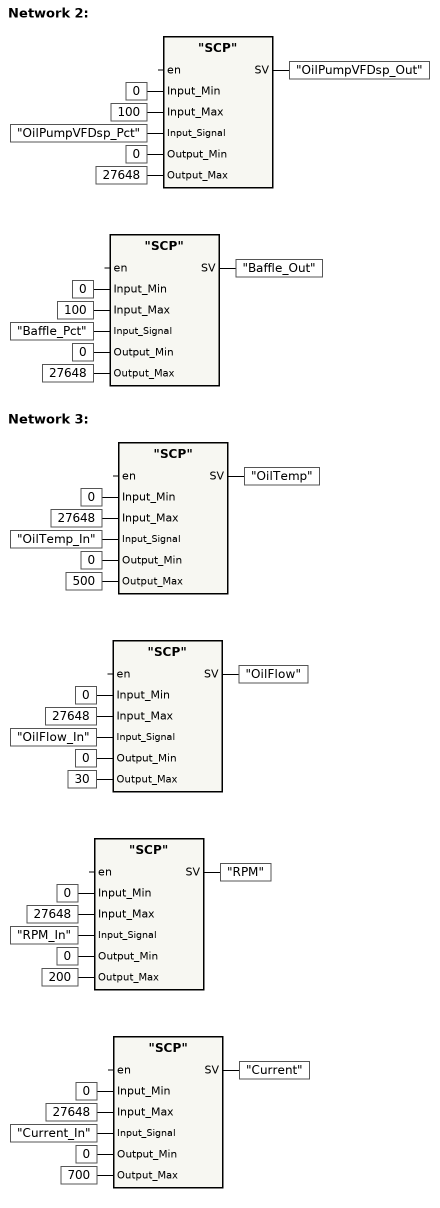
   "SCP"(Input_Min := 0,
         Input_Max := 100,
         Input_Signal := "OilPumpVFDsp_Pct",
         Output_Min := 0,
         Output_Max := 27648,
         SV => "OilPumpVFDsp_Out");
   "SCP"(Input_Min := 0,
         Input_Max := 100,
         Input_Signal := "Baffle_Pct",
         Output_Min := 0,
         Output_Max := 27648,
         SV => "Baffle_Out");
END_REGION

REGION Network 3
   // Analog Inputs
   "SCP"(Input_Min := 0,
         Input_Max := 27648,
         Input_Signal := "OilTemp_In",
         Output_Min := 0,
         Output_Max := 500,
         SV => "OilTemp");
   "SCP"(Input_Min := 0,
         Input_Max := 27648,
         Input_Signal := "OilFlow_In",
         Output_Min := 0,
         Output_Max := 30,
         SV => "OilFlow");
   "SCP"(Input_Min := 0,
         Input_Max := 27648,
         Input_Signal := "RPM_In",
         Output_Min := 0,
         Output_Max := 200,
         SV => "RPM");
   "SCP"(Input_Min := 0,
         Input_Max := 27648,
         Input_Signal := "Current_In",
         Output_Min := 0,
         Output_Max := 700,
         SV => "Current");
END_REGION

REGION Network 4: Full Auto Bit
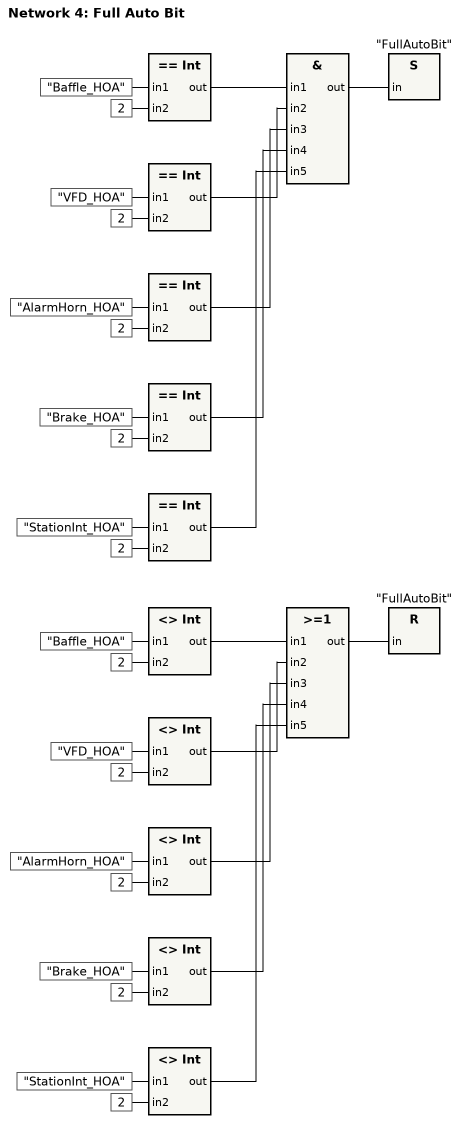
   IF ("Baffle_HOA" = 2) AND ("VFD_HOA" = 2) AND ("AlarmHorn_HOA" = 2) AND ("Brake_HOA" = 2) AND ("StationInt_HOA" = 2) THEN
       "FullAutoBit" := TRUE;
   END_IF;
   IF ("Baffle_HOA" <> 2) OR ("VFD_HOA" <> 2) OR ("AlarmHorn_HOA" <> 2) OR ("Brake_HOA" <> 2) OR ("StationInt_HOA" <> 2) THEN
       "FullAutoBit" := FALSE;
   END_IF;
END_REGION
END_FUNCTION_BLOCK

FUNCTION_BLOCK "IO_SCL"   // FB4, SCL
{ S7_Optimized_Access := 'TRUE' }
VERSION : 0.1
BEGIN
   // Digital Outputs
   IF "VFD_HOA" = 1 OR ("VFD_HOA" = 2 AND "OilPumpVFD_Ctrl") AND NOT "OilLowFlowAlarm" AND NOT "BrakeFailureAlarm" AND NOT "EStopAlarm" THEN
       "OilPumpVFDen_Out" := 1;
   ELSE
       "OilPumpVFDen_Out" := 0;
   END_IF;

   IF "Brake_HOA" = 1 OR ("Brake_HOA" = 2 AND "Brake_Ctrl") THEN
       "Brake_Out" := 1;
   ELSE
       "Brake_Out" := 0;
   END_IF;

   IF "AlarmHorn_HOA" = 1 OR ("AlarmHorn_HOA" = 2 AND "AlarmHorn_Ctrl") THEN
       "AlarmHorn_Out" := 1;
   ELSE
       "AlarmHorn_Out" := 0;
   END_IF;

   IF "StationInt_HOA" = 1 OR ("StationInt_HOA" = 2 AND "StationInt_Ctrl") AND NOT "BrakeFailureAlarm" AND NOT "EStopAlarm" THEN
       "StationInterlock_Out" := 1;
   ELSE
       "StationInterlock_Out" := 0;
   END_IF;

   IF "Baffle_HOA" = 1 OR ("Baffle_HOA" = 2 AND "Baffle_Ctrl") THEN
       "Baffle_En" := 1;
   ELSE
       "Baffle_En" := 0;
   END_IF;

   // Analog Outputs
   "SCP"(Input_Min:=0,
         Input_Max:=100,
         Input_Signal:="OilPumpVFDsp_Pct",
         Output_Min:=0,
         Output_Max:=27648,
         SV=>"OilPumpVFDsp_Out");
   "SCP"(Input_Min:=0,
         Input_Max:=100,
         Input_Signal:="Baffle_Pct",
         Output_Min:=0,
         Output_Max:=27648,
         SV=>"Baffle_Out");

   // Analog Inputs
   "SCP"(Input_Min := 0,
         Input_Max := 27648,
         Input_Signal := "OilTemp_In",
         Output_Min := 0,
         Output_Max := 500,
         SV => "OilTemp");
   "SCP"(Input_Min := 0,
         Input_Max := 27648,
         Input_Signal := "OilFlow_In",
         Output_Min := 0,
         Output_Max := 30,
         SV => "OilFlow");
   "SCP"(Input_Min := 0,
         Input_Max := 27648,
         Input_Signal := "RPM_In",
         Output_Min := 0,
         Output_Max := 200,
         SV => "RPM");
   "SCP"(Input_Min := 0,
         Input_Max := 27648,
         Input_Signal := "Current_In",
         Output_Min := 0,
         Output_Max := 700,
         SV => "Current");

   // Full Auto Bit
   IF "Baffle_HOA" = 2 AND "AlarmHorn_HOA" = 2 AND "VFD_HOA" = 2 AND "Brake_HOA" = 2 AND "StationInt_HOA" = 2 THEN
       "FullAutoBit" := 1;
   ELSE
       "FullAutoBit" := 0;
   END_IF;
END_FUNCTION_BLOCK

FUNCTION_BLOCK "IO_STL"   // FB5, STL
{ S7_Optimized_Access := 'TRUE' }
VERSION : 0.1
BEGIN

REGION Network 1
   // Digital Outputs
         A     "OilLowFlowAlarm";
         O     "BrakeFailureAlarm";
         O     "EStopAlarm";
         JC    ResetOilPumpVFD;
         CLR;
         L     "VFD_HOA";
         L     0;
         ==I;
         JC    ResetOilPumpVFD;
         CLR;
         L     "VFD_HOA";
         L     1;
         ==I;
         JC    SetOilPumpVFD;
         CLR;
         L     "VFD_HOA";
         L     2;
         ==I;
         JC    AutoOilPumpVFD;
         JU    Brake;

   AutoOilPumpVFD:A     "OilPumpVFD_Ctrl";
         JC    SetOilPumpVFD;
         JU    ResetOilPumpVFD;

   SetOilPumpVFD:S     "OilPumpVFDen_Out";
         JU    Brake;

   ResetOilPumpVFD:R     "OilPumpVFDen_Out";
         JU    Brake;

   Brake:L     "Brake_HOA";
         L     0;
         ==I;
         JC    ResetBrake;
         CLR;
         L     "Brake_HOA";
         L     1;
         ==I;
         JC    SetBrake;
         CLR;
         L     "Brake_HOA";
         L     2;
         ==I;
         JC    AutoBrake;
         JU    AlarmHorn;

   AutoBrake:A     "Brake_Ctrl";
         JC    SetBrake;
         JU    ResetBrake;

   SetBrake:S     "Brake_Out";
         JU    AlarmHorn;

   ResetBrake:R     "Brake_Out";
         JU    AlarmHorn;

   AlarmHorn:L     "AlarmHorn_HOA";
         L     0;
         ==I;
         JC    ResetAlarmHorn;
         CLR;
         L     "AlarmHorn_HOA";
         L     1;
         ==I;
         JC    SetAlarmHorn;
         CLR;
         L     "AlarmHorn_HOA";
         L     2;
         ==I;
         JC    AutoAlarmHorn;
         JU    StationInterlock;

   AutoAlarmHorn:A     "AlarmHorn_Ctrl";
         JC    SetAlarmHorn;
         JU    ResetAlarmHorn;

   SetAlarmHorn:S     "AlarmHorn_Out";
         JU    StationInterlock;

   ResetAlarmHorn:R     "AlarmHorn_Out";
         JU    StationInterlock;

   StationInterlock:A     "BrakeFailureAlarm";
         O     "EStopAlarm";
         JC    ResetStationInterlock;
         CLR;
         L     "StationInt_HOA";
         L     0;
         ==I;
         JC    ResetStationInterlock;
         CLR;
         L     "StationInt_HOA";
         L     1;
         ==I;
         JC    SetStationInterlock;
         CLR;
         L     "StationInt_HOA";
         L     2;
         ==I;
         JC    AutoStationInterlock;
         JU    Baffle;

   AutoStationInterlock:A     "StationInt_Ctrl";
         JC    SetStationInterlock;
         JU    ResetStationInterlock;

   SetStationInterlock:S     "StationInterlock_Out";
         JU    Baffle;

   ResetStationInterlock:R     "StationInterlock_Out";
         JU    Baffle;


   Baffle:L     "Baffle_HOA";
         L     0;
         ==I;
         JC    ResetBaffle;
         CLR;
         L     "Baffle_HOA";
         L     1;
         ==I;
         JC    SetBaffle;
         CLR;
         L     "Baffle_HOA";
         L     2;
         ==I;
         JC    AutoBaffle;
         JU    AnalogOutputs;

   AutoBaffle:A     "Baffle_Ctrl";
         JC    SetBaffle;
         JU    ResetBaffle;

   SetBaffle:S     "Baffle_En";
         JU    AnalogOutputs;

   ResetBaffle:R     "Baffle_En";
         JU    AnalogOutputs;
END_REGION

REGION Network 2
   // Analog Outputs
   AnalogOutputs:CALL  "SCP"
         ( Input_Min    := 0,
           Input_Max    := 100,
           Input_Signal := "OilPumpVFDsp_Pct",
           Output_Min   := 0,
           Output_Max   := 27648,
           SV           := "OilPumpVFDsp_Out"
         );
         CALL  "SCP"
         ( Input_Min    := 0,
           Input_Max    := 100,
           Input_Signal := "Baffle_Pct",
           Output_Min   := 0,
           Output_Max   := 27648,
           SV           := "Baffle_Out"
         );
END_REGION

REGION Network 3
   // Analog Inputs
   AnalogInputs:CALL  "SCP"
         ( Input_Min    := 0,
           Input_Max    := 27648,
           Input_Signal := "OilTemp_In",
           Output_Min   := 0,
           Output_Max   := 500,
           SV           := "OilTemp"
         );
         CALL  "SCP"
         ( Input_Min    := 0,
           Input_Max    := 27648,
           Input_Signal := "OilFlow_In",
           Output_Min   := 0,
           Output_Max   := 30,
           SV           := "OilFlow"
         );
         CALL  "SCP"
         ( Input_Min    := 0,
           Input_Max    := 27648,
           Input_Signal := "RPM_In",
           Output_Min   := 0,
           Output_Max   := 200,
           SV           := "RPM"
         );
         CALL  "SCP"
         ( Input_Min    := 0,
           Input_Max    := 27648,
           Input_Signal := "Current_In",
           Output_Min   := 0,
           Output_Max   := 700,
           SV           := "Current"
         );
END_REGION

REGION Network 4: Full Auto Bit
         CLR;
         L     "Baffle_HOA";
         L     2;
         ==I;
         NOT;
         JC    ResetFullAuto;
         CLR;
         L     "AlarmHorn_HOA";
         L     2;
         ==I;
         NOT;
         JC    ResetFullAuto;
         CLR;
         L     "Brake_HOA";
         L     2;
         ==I;
         NOT;
         JC    ResetFullAuto;
         CLR;
         L     "VFD_HOA";
         L     2;
         ==I;
         NOT;
         JC    ResetFullAuto;
         CLR;
         L     "StationInt_HOA";
         L     2;
         ==I;
         NOT;
         JC    ResetFullAuto;
         CLR;
         SET;
         S     "FullAutoBit";
         JU    EndOfLine;

   ResetFullAuto:SET;
         NOT;
         R     "FullAutoBit";
         JU    EndOfLine;

   EndOfLine:BE;
END_REGION
END_FUNCTION_BLOCK

FUNCTION_BLOCK "HOA_LAD"   // FB6, LAD
{ S7_Optimized_Access := 'TRUE' }
VERSION : 0.1
   VAR
      OS1 : Bool;
      OS2 : Bool;
      OS3 : Bool;
      OS4 : Bool;
      OS5 : Bool;
      OS6 : Bool;
      OS7 : Bool;
      OS8 : Bool;
      OS9 : Bool;
      OS10 : Bool;
      OS11 : Bool;
      OS12 : Bool;
   END_VAR
   VAR_TEMP   // added for the SCL form of the ladder/FBD networks
      _w1 : Bool;
      _w2 : Bool;
      _w3 : Bool;
   END_VAR
BEGIN

REGION Network 1
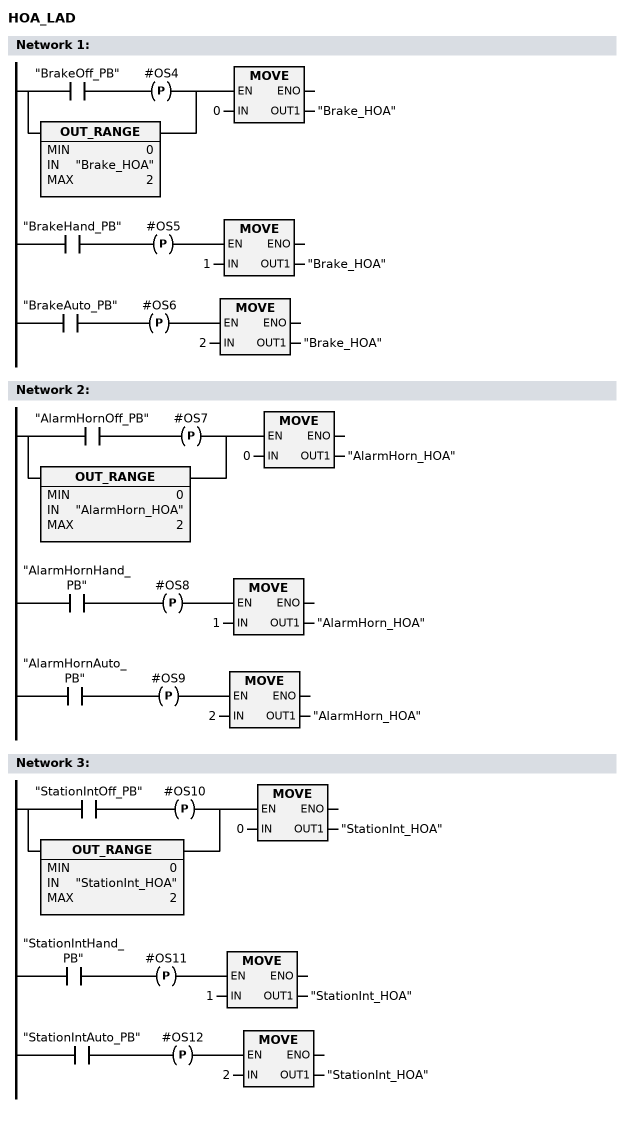
   #_w1 := "BrakeOff_PB" AND NOT #OS4;   // rising edge
   #OS4 := "BrakeOff_PB";
   IF #_w1 OR ("Brake_HOA" < 0) OR ("Brake_HOA" > 2) THEN "Brake_HOA" := 0; END_IF;
   #_w2 := "BrakeHand_PB" AND NOT #OS5;   // rising edge
   #OS5 := "BrakeHand_PB";
   IF #_w2 THEN "Brake_HOA" := 1; END_IF;
   #_w3 := "BrakeAuto_PB" AND NOT #OS6;   // rising edge
   #OS6 := "BrakeAuto_PB";
   IF #_w3 THEN "Brake_HOA" := 2; END_IF;
END_REGION

REGION Network 2
   #_w1 := "AlarmHornOff_PB" AND NOT #OS7;   // rising edge
   #OS7 := "AlarmHornOff_PB";
   IF #_w1 OR ("AlarmHorn_HOA" < 0) OR ("AlarmHorn_HOA" > 2) THEN "AlarmHorn_HOA" := 0; END_IF;
   #_w2 := "AlarmHornHand_PB" AND NOT #OS8;   // rising edge
   #OS8 := "AlarmHornHand_PB";
   IF #_w2 THEN "AlarmHorn_HOA" := 1; END_IF;
   #_w3 := "AlarmHornAuto_PB" AND NOT #OS9;   // rising edge
   #OS9 := "AlarmHornAuto_PB";
   IF #_w3 THEN "AlarmHorn_HOA" := 2; END_IF;
END_REGION

REGION Network 3
   #_w1 := "StationIntOff_PB" AND NOT #OS10;   // rising edge
   #OS10 := "StationIntOff_PB";
   IF #_w1 OR ("StationInt_HOA" < 0) OR ("StationInt_HOA" > 2) THEN "StationInt_HOA" := 0; END_IF;
   #_w2 := "StationIntHand_PB" AND NOT #OS11;   // rising edge
   #OS11 := "StationIntHand_PB";
   IF #_w2 THEN "StationInt_HOA" := 1; END_IF;
   #_w3 := "StationIntAuto_PB" AND NOT #OS12;   // rising edge
   #OS12 := "StationIntAuto_PB";
   IF #_w3 THEN "StationInt_HOA" := 2; END_IF;
END_REGION
END_FUNCTION_BLOCK

FUNCTION_BLOCK "HOA_FBD"   // FB7, FBD
{ S7_Optimized_Access := 'TRUE' }
VERSION : 0.1
   VAR
      ON1 : Bool;
      ON2 : Bool;
      ON3 : Bool;
      ON4 : Bool;
      ON5 : Bool;
      ON6 : Bool;
      ON7 : Bool;
      ON8 : Bool;
      ON9 : Bool;
      ON10 : Bool;
      ON11 : Bool;
      ON12 : Bool;
   END_VAR
   VAR_TEMP   // added for the SCL form of the ladder/FBD networks
      _w1 : Bool;
      _w2 : Bool;
      _w3 : Bool;
   END_VAR
BEGIN

REGION Network 1
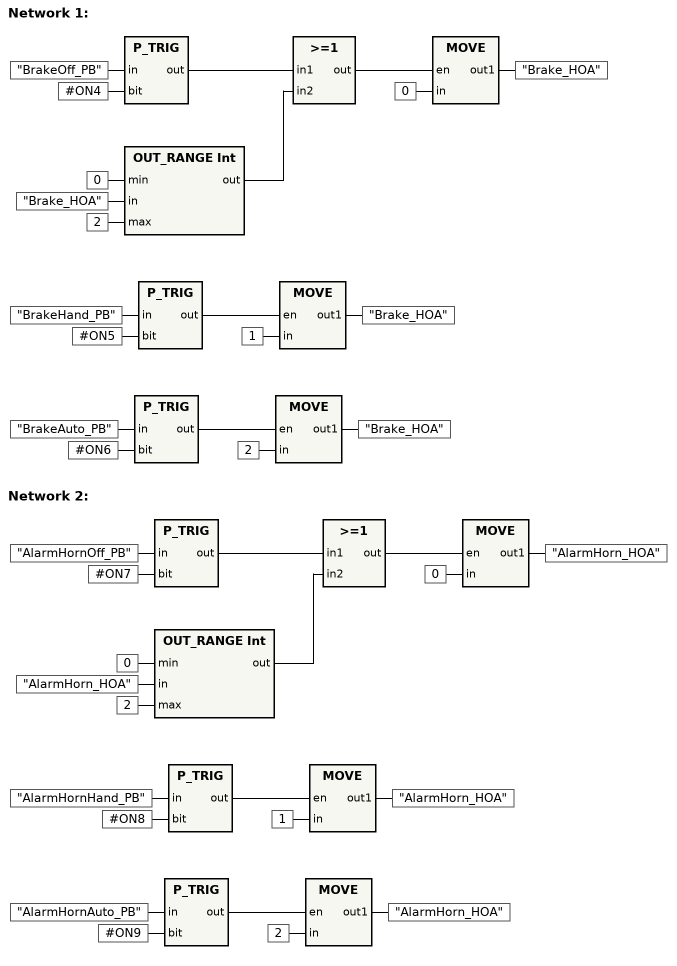
   #_w1 := "BrakeOff_PB" AND NOT #ON4;   // rising edge
   #ON4 := "BrakeOff_PB";
   IF #_w1 OR ("Brake_HOA" < 0) OR ("Brake_HOA" > 2) THEN "Brake_HOA" := 0; END_IF;
   #_w2 := "BrakeHand_PB" AND NOT #ON5;   // rising edge
   #ON5 := "BrakeHand_PB";
   IF #_w2 THEN "Brake_HOA" := 1; END_IF;
   #_w3 := "BrakeAuto_PB" AND NOT #ON6;   // rising edge
   #ON6 := "BrakeAuto_PB";
   IF #_w3 THEN "Brake_HOA" := 2; END_IF;
END_REGION

REGION Network 2
   #_w1 := "AlarmHornOff_PB" AND NOT #ON7;   // rising edge
   #ON7 := "AlarmHornOff_PB";
   IF #_w1 OR ("AlarmHorn_HOA" < 0) OR ("AlarmHorn_HOA" > 2) THEN "AlarmHorn_HOA" := 0; END_IF;
   #_w2 := "AlarmHornHand_PB" AND NOT #ON8;   // rising edge
   #ON8 := "AlarmHornHand_PB";
   IF #_w2 THEN "AlarmHorn_HOA" := 1; END_IF;
   #_w3 := "AlarmHornAuto_PB" AND NOT #ON9;   // rising edge
   #ON9 := "AlarmHornAuto_PB";
   IF #_w3 THEN "AlarmHorn_HOA" := 2; END_IF;
END_REGION

REGION Network 3
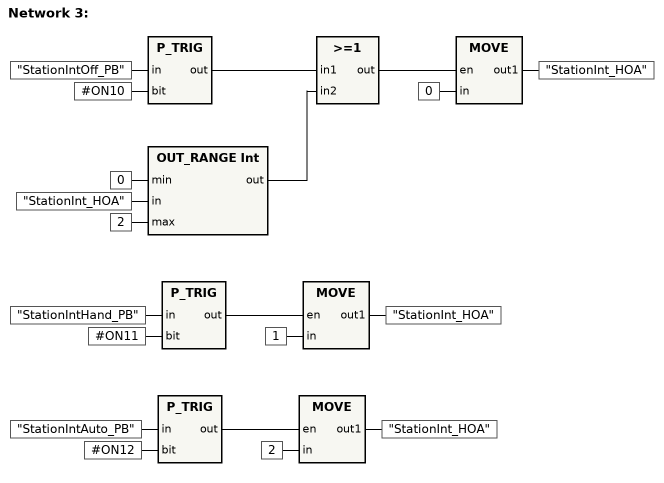
   #_w1 := "StationIntOff_PB" AND NOT #ON10;   // rising edge
   #ON10 := "StationIntOff_PB";
   IF #_w1 OR ("StationInt_HOA" < 0) OR ("StationInt_HOA" > 2) THEN "StationInt_HOA" := 0; END_IF;
   #_w2 := "StationIntHand_PB" AND NOT #ON11;   // rising edge
   #ON11 := "StationIntHand_PB";
   IF #_w2 THEN "StationInt_HOA" := 1; END_IF;
   #_w3 := "StationIntAuto_PB" AND NOT #ON12;   // rising edge
   #ON12 := "StationIntAuto_PB";
   IF #_w3 THEN "StationInt_HOA" := 2; END_IF;
END_REGION
END_FUNCTION_BLOCK

FUNCTION_BLOCK "HOA_SCL"   // FB8, SCL
{ S7_Optimized_Access := 'TRUE' }
VERSION : 0.1
BEGIN
   // Brake HOA Controls
   IF "BrakeOff_PB" AND "Brake_HOA" <> 0 OR "Brake_HOA" < 0 OR "Brake_HOA" > 2 THEN
       "Brake_HOA" := 0;
   END_IF;

   IF "BrakeHand_PB" AND "Brake_HOA" <> 1 THEN
       "Brake_HOA" := 1;
   END_IF;

   IF "BrakeAuto_PB" AND "Brake_HOA" <> 2 THEN
       "Brake_HOA" := 2;
   END_IF;

   // Alarm Horn HOA Controls
   IF "AlarmHornOff_PB" AND "AlarmHorn_HOA" <> 0 OR "AlarmHorn_HOA" < 0 OR "AlarmHorn_HOA" > 2 THEN
       "AlarmHorn_HOA" := 0;
   END_IF;

   IF "AlarmHornHand_PB" AND "AlarmHorn_HOA" <> 1 THEN
       "AlarmHorn_HOA" := 1;
   END_IF;

   IF "AlarmHornAuto_PB" AND "AlarmHorn_HOA" <> 2 THEN
       "AlarmHorn_HOA" := 2;
   END_IF;

   // Station Interlock HOA Controls
   IF "StationIntOff_PB" AND "StationInt_HOA" <> 0 OR "StationInt_HOA" < 0 OR "StationInt_HOA" > 2 THEN
       "StationInt_HOA" := 0;
   END_IF;

   IF "StationIntHand_PB" AND "StationInt_HOA" <> 1 THEN
       "StationInt_HOA" := 1;
   END_IF;

   IF "StationIntAuto_PB" AND "StationInt_HOA" <> 2 THEN
       "StationInt_HOA" := 2;
   END_IF;
END_FUNCTION_BLOCK

FUNCTION_BLOCK "HOA_STL"   // FB9, STL
{ S7_Optimized_Access := 'TRUE' }
VERSION : 0.1
   VAR
      OS1 : Bool;
      OS2 : Bool;
      OS3 : Bool;
      OS4 : Bool;
      OS5 : Bool;
      OS6 : Bool;
      OS7 : Bool;
      OS8 : Bool;
      OS9 : Bool;
      OS10 : Bool;
      OS11 : Bool;
      OS12 : Bool;
   END_VAR
BEGIN

REGION Network 1
         L     "Brake_HOA";
         L     0;
         <I;
         JC    SetBrake_HOA0;
         CLR;
         L     "Brake_HOA";
         L     2;
         >I;
         JC    SetBrake_HOA0;
         CLR;
         A     "BrakeOff_PB";
         FP    #OS4;
         JC    SetBrake_HOA0;
         CLR;
         A     "BrakeHand_PB";
         FP    #OS5;
         JC    SetBrake_HOA1;
         CLR;
         A     "BrakeAuto_PB";
         FP    #OS6;
         JC    SetBrake_HOA2;
         JU    AlarmHorn;

   SetBrake_HOA0:L     0;
         T     "Brake_HOA";
         JU    AlarmHorn;

   SetBrake_HOA1:L     1;
         T     "Brake_HOA";
         JU    AlarmHorn;

   SetBrake_HOA2:L     2;
         T     "Brake_HOA";
         JU    AlarmHorn;

   AlarmHorn:L     "AlarmHorn_HOA";
         L     0;
         <I;
         JC    SetAlarmHorn_HOA0;
         CLR;
         L     "AlarmHorn_HOA";
         L     2;
         >I;
         JC    SetAlarmHorn_HOA0;
         CLR;
         A     "AlarmHornOff_PB";
         FP    #OS7;
         JC    SetAlarmHorn_HOA0;
         CLR;
         A     "AlarmHornHand_PB";
         FP    #OS8;
         JC    SetAlarmHorn_HOA1;
         CLR;
         A     "AlarmHornAuto_PB";
         FP    #OS9;
         JC    SetAlarmHorn_HOA2;
         JU    StationInterlock;

   SetAlarmHorn_HOA0:L     0;
         T     "AlarmHorn_HOA";
         JU    StationInterlock;

   SetAlarmHorn_HOA1:L     1;
         T     "AlarmHorn_HOA";
         JU    StationInterlock;

   SetAlarmHorn_HOA2:L     2;
         T     "AlarmHorn_HOA";
         JU    StationInterlock;

   StationInterlock:L     "StationInt_HOA";
         L     0;
         <I;
         JC    SetStationInterlock_HOA0;
         CLR;
         L     "StationInt_HOA";
         L     2;
         >I;
         JC    SetStationInterlock_HOA0;
         CLR;
         A     "StationIntOff_PB";
         FP    #OS10;
         JC    SetStationInterlock_HOA0;
         CLR;
         A     "StationIntHand_PB";
         FP    #OS11;
         JC    SetStationInterlock_HOA1;
         CLR;
         A     "StationIntAuto_PB";
         FP    #OS12;
         JC    SetStationInterlock_HOA2;
         JU    EndOfLine;

   SetStationInterlock_HOA0:L     0;
         T     "StationInt_HOA";
         JU    EndOfLine;

   SetStationInterlock_HOA1:L     1;
         T     "StationInt_HOA";
         JU    EndOfLine;

   SetStationInterlock_HOA2:L     2;
         T     "StationInt_HOA";
         JU    EndOfLine;

   EndOfLine:BE;
END_REGION
END_FUNCTION_BLOCK

FUNCTION_BLOCK "ALARMS_LAD"   // FB10, LAD
{ S7_Optimized_Access := 'TRUE' }
VERSION : 0.1
   VAR
      OS1 : Bool;
      OS2 : Bool;
      OS3 : Bool;
      OS4 : Bool;
      OS5 : Bool;
      OS6 : Bool;
      OS7 : Bool;
      OS8 : Bool;
      OS9 : Bool;
      OS10 : Bool;
   END_VAR
   VAR_TEMP
      OLFD : Int;
      OLFAT : Bool;
      TV1 : Time;
      OCD : Int;
      TV2 : Time;
      OCAT : Bool;
      HOTD : Int;
      TV3 : Time;
      HOTAT : Bool;
      ROSD : Int;
      TV4 : Time;
      ROSAT : Bool;
      OHFD : Int;
      TV5 : Time;
      OHFAT : Bool;
      BFD : Int;
      TV6 : Time;
      BFAT : Bool;
      ESAT : Bool;
      AlarmHornTrigger : Bool;
   END_VAR
   VAR_TEMP   // added for the SCL form of the ladder/FBD networks
      _w1 : Bool;
      _w2 : Bool;
   END_VAR
BEGIN

REGION Network 1
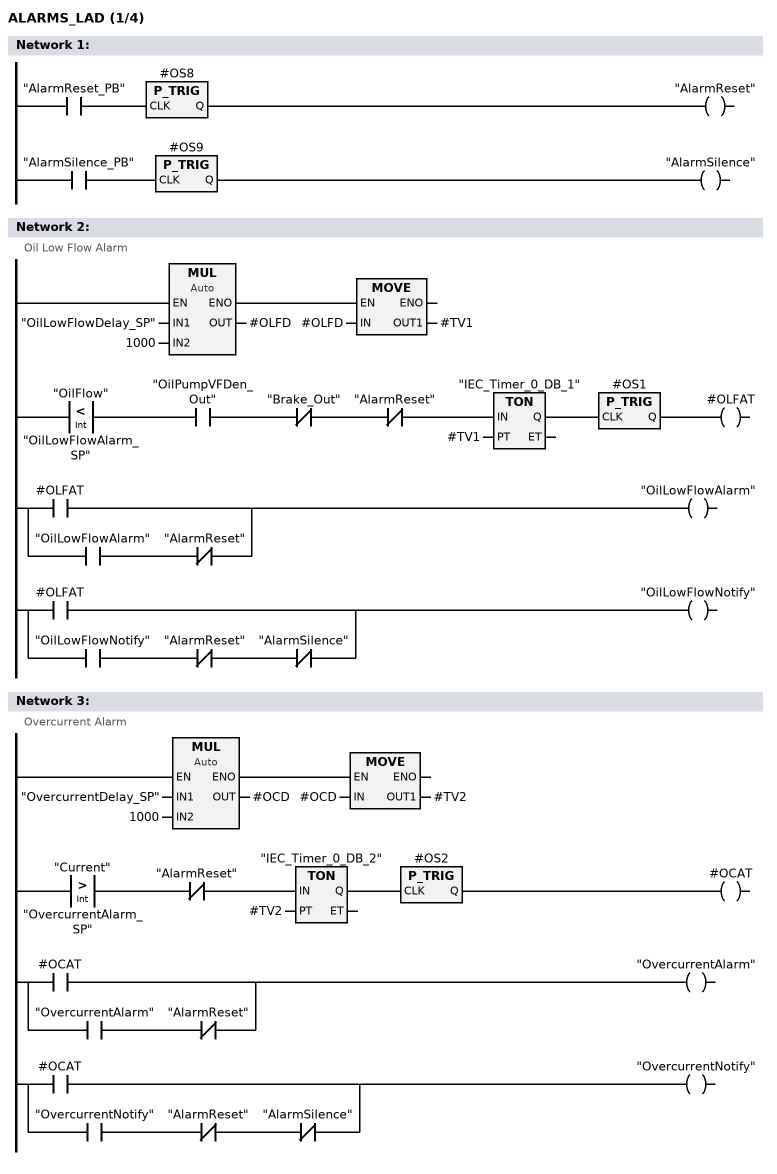
   RUNG wire#powerrail
      Contact( "AlarmReset_PB" )
      P_Trig( #OS8 )
      Coil( "AlarmReset" )
   END_RUNG
   RUNG wire#powerrail
      Contact( "AlarmSilence_PB" )
      P_Trig( #OS9 )
      Coil( "AlarmSilence" )
   END_RUNG
   // the same network as SCL:
   #_w1 := "AlarmReset_PB" AND NOT #OS8;   // rising edge
   #OS8 := "AlarmReset_PB";
   "AlarmReset" := #_w1;
   #_w2 := "AlarmSilence_PB" AND NOT #OS9;   // rising edge
   #OS9 := "AlarmSilence_PB";
   "AlarmSilence" := #_w2;
END_REGION

REGION Network 2
   // Oil Low Flow Alarm
   #OLFD := "OilLowFlowDelay_SP" * 1000;
   #TV1 := #OLFD;
   "IEC_Timer_0_DB_1".TON(IN := ("OilFlow" < "OilLowFlowAlarm_SP") AND "OilPumpVFDen_Out" AND NOT "Brake_Out" AND NOT "AlarmReset",
                          PT := #TV1);
   #_w1 := "IEC_Timer_0_DB_1".Q AND NOT #OS1;   // rising edge
   #OS1 := "IEC_Timer_0_DB_1".Q;
   #OLFAT := #_w1;
   "OilLowFlowAlarm" := #OLFAT OR ("OilLowFlowAlarm" AND NOT "AlarmReset");
   "OilLowFlowNotify" := #OLFAT OR ("OilLowFlowNotify" AND NOT "AlarmReset" AND NOT "AlarmSilence");
END_REGION

REGION Network 3
   // Overcurrent Alarm
   #OCD := "OvercurrentDelay_SP" * 1000;
   #TV2 := #OCD;
   "IEC_Timer_0_DB_2".TON(IN := ("Current" > "OvercurrentAlarm_SP") AND NOT "AlarmReset", PT := #TV2);
   #_w1 := "IEC_Timer_0_DB_2".Q AND NOT #OS2;   // rising edge
   #OS2 := "IEC_Timer_0_DB_2".Q;
   #OCAT := #_w1;
   "OvercurrentAlarm" := #OCAT OR ("OvercurrentAlarm" AND NOT "AlarmReset");
   "OvercurrentNotify" := #OCAT OR ("OvercurrentNotify" AND NOT "AlarmReset" AND NOT "AlarmSilence");
END_REGION

REGION Network 4
   // High Oil Temp Alarm
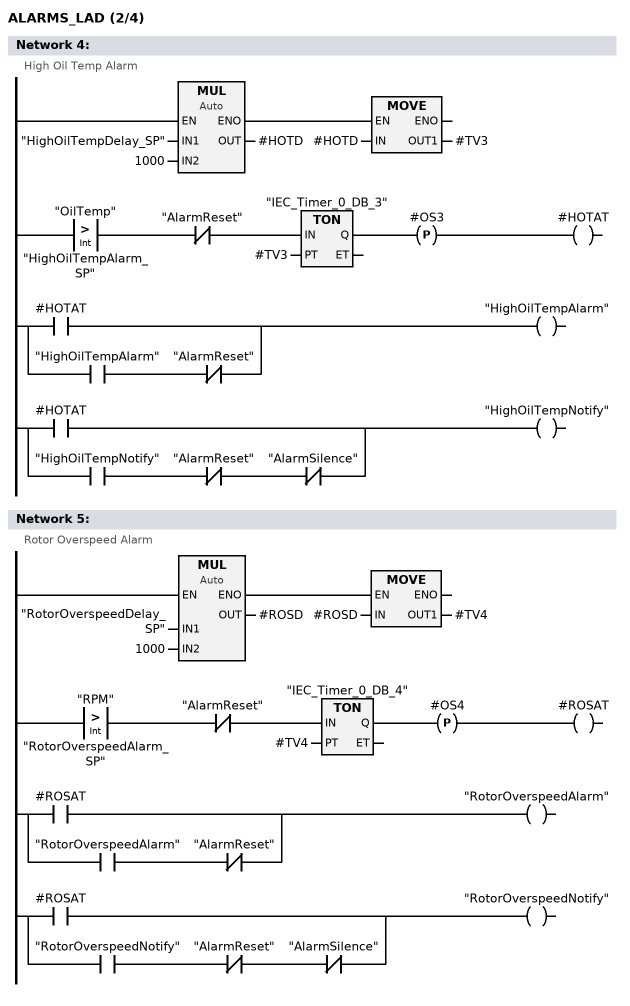
   #HOTD := "HighOilTempDelay_SP" * 1000;
   #TV3 := #HOTD;
   "IEC_Timer_0_DB_3".TON(IN := ("OilTemp" > "HighOilTempAlarm_SP") AND NOT "AlarmReset", PT := #TV3);
   #_w1 := "IEC_Timer_0_DB_3".Q AND NOT #OS3;   // rising edge
   #OS3 := "IEC_Timer_0_DB_3".Q;
   #HOTAT := #_w1;
   "HighOilTempAlarm" := #HOTAT OR ("HighOilTempAlarm" AND NOT "AlarmReset");
   "HighOilTempNotify" := #HOTAT OR ("HighOilTempNotify" AND NOT "AlarmReset" AND NOT "AlarmSilence");
END_REGION

REGION Network 5
   // Rotor Overspeed Alarm
   #ROSD := "RotorOverspeedDelay_SP" * 1000;
   #TV4 := #ROSD;
   "IEC_Timer_0_DB_4".TON(IN := ("RPM" > "RotorOverspeedAlarm_SP") AND NOT "AlarmReset", PT := #TV4);
   #_w1 := "IEC_Timer_0_DB_4".Q AND NOT #OS4;   // rising edge
   #OS4 := "IEC_Timer_0_DB_4".Q;
   #ROSAT := #_w1;
   "RotorOverspeedAlarm" := #ROSAT OR ("RotorOverspeedAlarm" AND NOT "AlarmReset");
   "RotorOverspeedNotify" := #ROSAT OR ("RotorOverspeedNotify" AND NOT "AlarmReset" AND NOT "AlarmSilence");
END_REGION

REGION Network 6
   // Oil High Flow Alarm
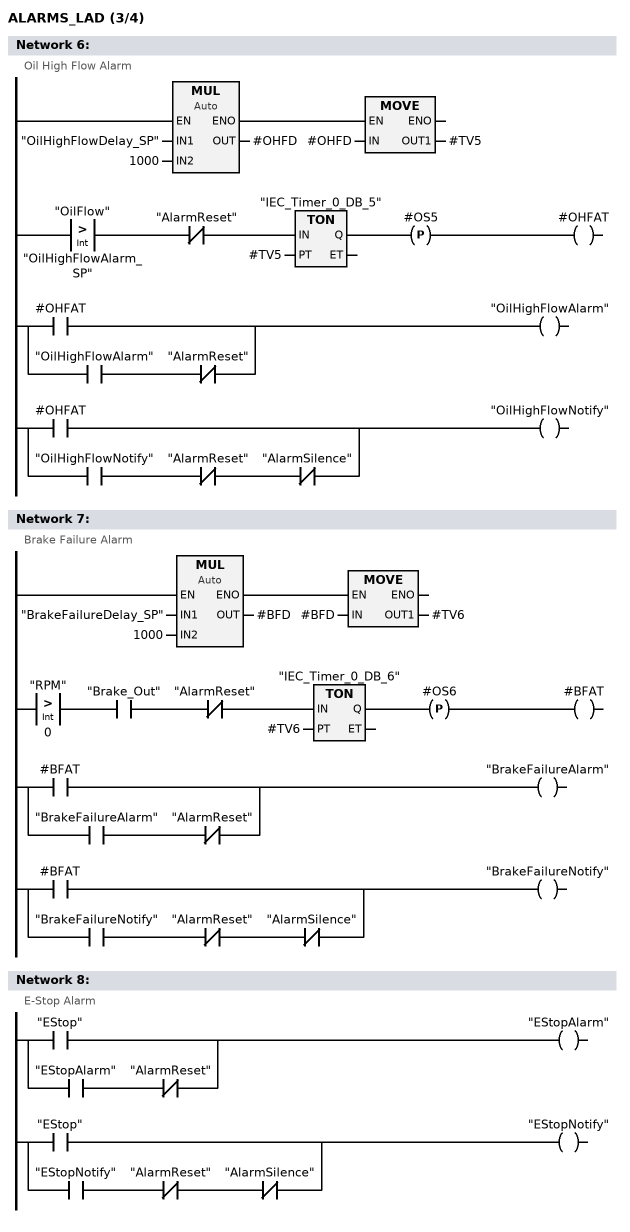
   #OHFD := "OilHighFlowDelay_SP" * 1000;
   #TV5 := #OHFD;
   "IEC_Timer_0_DB_5".TON(IN := ("OilFlow" > "OilHighFlowAlarm_SP") AND NOT "AlarmReset", PT := #TV5);
   #_w1 := "IEC_Timer_0_DB_5".Q AND NOT #OS5;   // rising edge
   #OS5 := "IEC_Timer_0_DB_5".Q;
   #OHFAT := #_w1;
   "OilHighFlowAlarm" := #OHFAT OR ("OilHighFlowAlarm" AND NOT "AlarmReset");
   "OilHighFlowNotify" := #OHFAT OR ("OilHighFlowNotify" AND NOT "AlarmReset" AND NOT "AlarmSilence");
END_REGION

REGION Network 7
   // Brake Failure Alarm
   #BFD := "BrakeFailureDelay_SP" * 1000;
   #TV6 := #BFD;
   "IEC_Timer_0_DB_6".TON(IN := ("RPM" > 0) AND "Brake_Out" AND NOT "AlarmReset", PT := #TV6);
   #_w1 := "IEC_Timer_0_DB_6".Q AND NOT #OS6;   // rising edge
   #OS6 := "IEC_Timer_0_DB_6".Q;
   #BFAT := #_w1;
   "BrakeFailureAlarm" := #BFAT OR ("BrakeFailureAlarm" AND NOT "AlarmReset");
   "BrakeFailureNotify" := #BFAT OR ("BrakeFailureNotify" AND NOT "AlarmReset" AND NOT "AlarmSilence");
END_REGION

REGION Network 8
   // E-Stop Alarm
   RUNG wire#powerrail
      Contact( "EStop" )
      wire#w1
      Coil( "EStopAlarm" )
   END_RUNG
   RUNG wire#powerrail
      Contact( "EStopAlarm" )
      I_Contact( "AlarmReset" )
   END_RUNG wire#w1
   RUNG wire#powerrail
      Contact( "EStop" )
      wire#w2
      Coil( "EStopNotify" )
   END_RUNG
   RUNG wire#powerrail
      Contact( "EStopNotify" )
      I_Contact( "AlarmReset" )
      I_Contact( "AlarmSilence" )
   END_RUNG wire#w2
   // the same network as SCL:
   "EStopAlarm" := "EStop" OR ("EStopAlarm" AND NOT "AlarmReset");
   "EStopNotify" := "EStop" OR ("EStopNotify" AND NOT "AlarmReset" AND NOT "AlarmSilence");
END_REGION

REGION Network 9
   // Alarm Horn Control
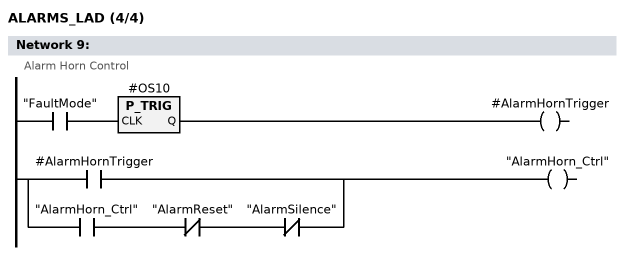
   RUNG wire#powerrail
      Contact( "FaultMode" )
      P_Trig( #OS10 )
      Coil( #AlarmHornTrigger )
   END_RUNG
   RUNG wire#powerrail
      Contact( #AlarmHornTrigger )
      wire#w1
      Coil( "AlarmHorn_Ctrl" )
   END_RUNG
   RUNG wire#powerrail
      Contact( "AlarmHorn_Ctrl" )
      I_Contact( "AlarmReset" )
      I_Contact( "AlarmSilence" )
   END_RUNG wire#w1
   // the same network as SCL:
   #_w1 := "FaultMode" AND NOT #OS10;   // rising edge
   #OS10 := "FaultMode";
   #AlarmHornTrigger := #_w1;
   "AlarmHorn_Ctrl" := #AlarmHornTrigger OR ("AlarmHorn_Ctrl" AND NOT "AlarmReset" AND NOT "AlarmSilence");
END_REGION
END_FUNCTION_BLOCK

FUNCTION_BLOCK "ALARMS_FBD"   // FB11, FBD
{ S7_Optimized_Access := 'TRUE' }
VERSION : 0.1
   VAR
      OS1 : Bool;
      OS2 : Bool;
      OS3 : Bool;
      OS4 : Bool;
      OS5 : Bool;
      OS6 : Bool;
      OS7 : Bool;
      OS8 : Bool;
      OS9 : Bool;
      OS10 : Bool;
   END_VAR
   VAR_TEMP
      OLFD : Int;
      TV1 : Time;
      OLFAT : Bool;
      OCD : Int;
      TV2 : Time;
      OCAT : Bool;
      HOTD : Int;
      TV3 : Time;
      HOTAT : Bool;
      ROSD : Int;
      TV4 : Time;
      ROSAT : Bool;
      OHFD : Int;
      TV5 : Time;
      OHFAT : Bool;
      BFD : Int;
      TV6 : Time;
      BFAT : Bool;
      ESAT : Bool;
   END_VAR
   VAR_TEMP   // added for the SCL form of the ladder/FBD networks
      _w1 : Bool;
      _w2 : Bool;
   END_VAR
BEGIN

REGION Network 1
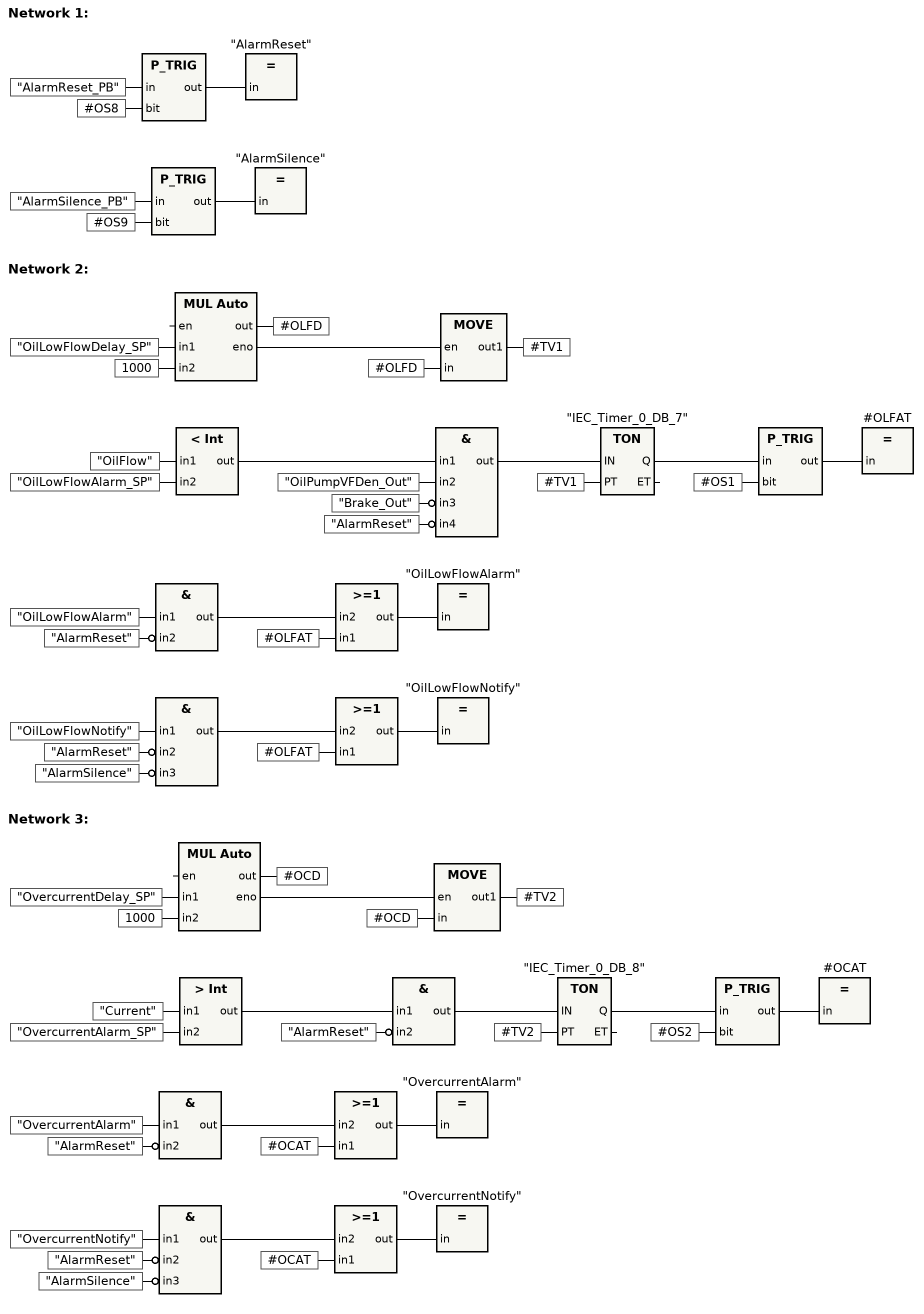
   #_w1 := "AlarmReset_PB" AND NOT #OS8;   // rising edge
   #OS8 := "AlarmReset_PB";
   "AlarmReset" := #_w1;
   #_w2 := "AlarmSilence_PB" AND NOT #OS9;   // rising edge
   #OS9 := "AlarmSilence_PB";
   "AlarmSilence" := #_w2;
END_REGION

REGION Network 2
   // Oil Low Flow Alarm
   #OLFD := "OilLowFlowDelay_SP" * 1000;
   #TV1 := #OLFD;
   "IEC_Timer_0_DB_7".TON(IN := ("OilFlow" < "OilLowFlowAlarm_SP") AND "OilPumpVFDen_Out" AND NOT "Brake_Out" AND NOT "AlarmReset",
                          PT := #TV1);
   #_w1 := "IEC_Timer_0_DB_7".Q AND NOT #OS1;   // rising edge
   #OS1 := "IEC_Timer_0_DB_7".Q;
   #OLFAT := #_w1;
   "OilLowFlowAlarm" := ("OilLowFlowAlarm" AND NOT "AlarmReset") OR #OLFAT;
   "OilLowFlowNotify" := ("OilLowFlowNotify" AND NOT "AlarmReset" AND NOT "AlarmSilence") OR #OLFAT;
END_REGION

REGION Network 3
   // Overcurrent Alarm
   #OCD := "OvercurrentDelay_SP" * 1000;
   #TV2 := #OCD;
   "IEC_Timer_0_DB_8".TON(IN := ("Current" > "OvercurrentAlarm_SP") AND NOT "AlarmReset", PT := #TV2);
   #_w1 := "IEC_Timer_0_DB_8".Q AND NOT #OS2;   // rising edge
   #OS2 := "IEC_Timer_0_DB_8".Q;
   #OCAT := #_w1;
   "OvercurrentAlarm" := ("OvercurrentAlarm" AND NOT "AlarmReset") OR #OCAT;
   "OvercurrentNotify" := ("OvercurrentNotify" AND NOT "AlarmReset" AND NOT "AlarmSilence") OR #OCAT;
END_REGION

REGION Network 4
   // High Oil Temp Alarm
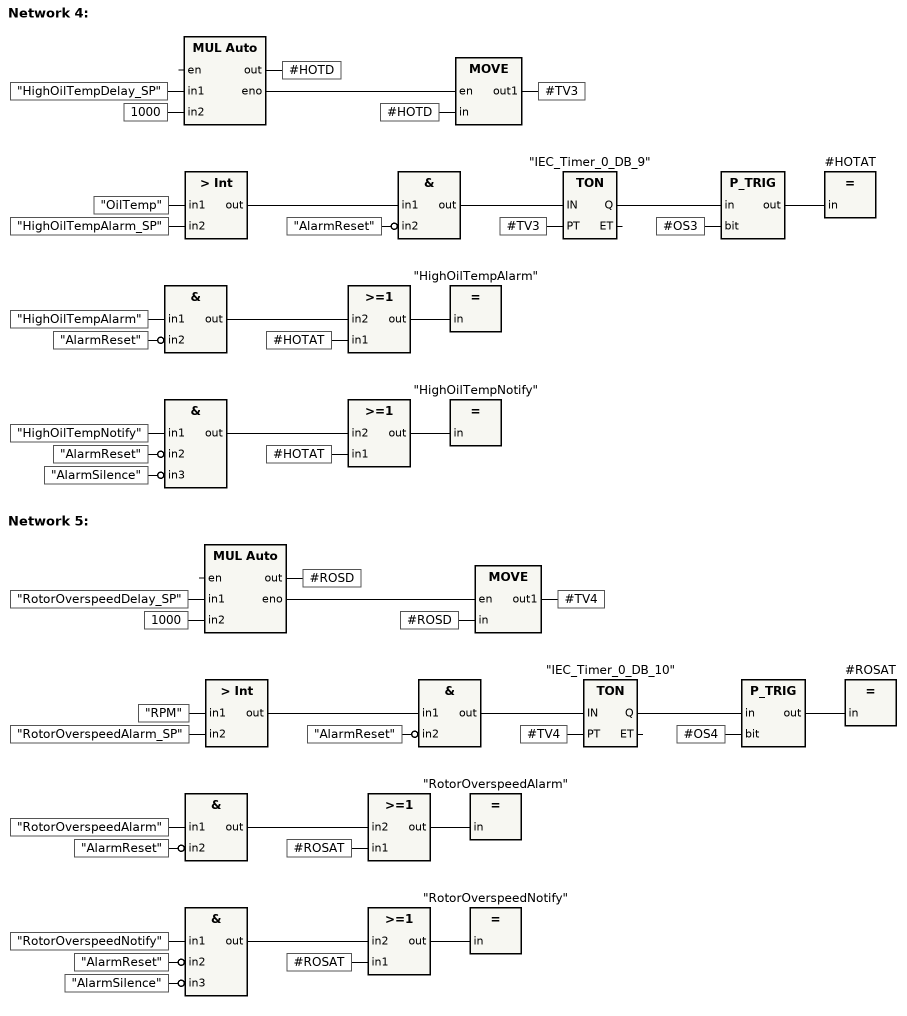
   #HOTD := "HighOilTempDelay_SP" * 1000;
   #TV3 := #HOTD;
   "IEC_Timer_0_DB_9".TON(IN := ("OilTemp" > "HighOilTempAlarm_SP") AND NOT "AlarmReset", PT := #TV3);
   #_w1 := "IEC_Timer_0_DB_9".Q AND NOT #OS3;   // rising edge
   #OS3 := "IEC_Timer_0_DB_9".Q;
   #HOTAT := #_w1;
   "HighOilTempAlarm" := ("HighOilTempAlarm" AND NOT "AlarmReset") OR #HOTAT;
   "HighOilTempNotify" := ("HighOilTempNotify" AND NOT "AlarmReset" AND NOT "AlarmSilence") OR #HOTAT;
END_REGION

REGION Network 5
   // Rotor Overspeed Alarm
   #ROSD := "RotorOverspeedDelay_SP" * 1000;
   #TV4 := #ROSD;
   "IEC_Timer_0_DB_10".TON(IN := ("RPM" > "RotorOverspeedAlarm_SP") AND NOT "AlarmReset", PT := #TV4);
   #_w1 := "IEC_Timer_0_DB_10".Q AND NOT #OS4;   // rising edge
   #OS4 := "IEC_Timer_0_DB_10".Q;
   #ROSAT := #_w1;
   "RotorOverspeedAlarm" := ("RotorOverspeedAlarm" AND NOT "AlarmReset") OR #ROSAT;
   "RotorOverspeedNotify" := ("RotorOverspeedNotify" AND NOT "AlarmReset" AND NOT "AlarmSilence") OR #ROSAT;
END_REGION

REGION Network 6
   // Oil High Flow Alarm
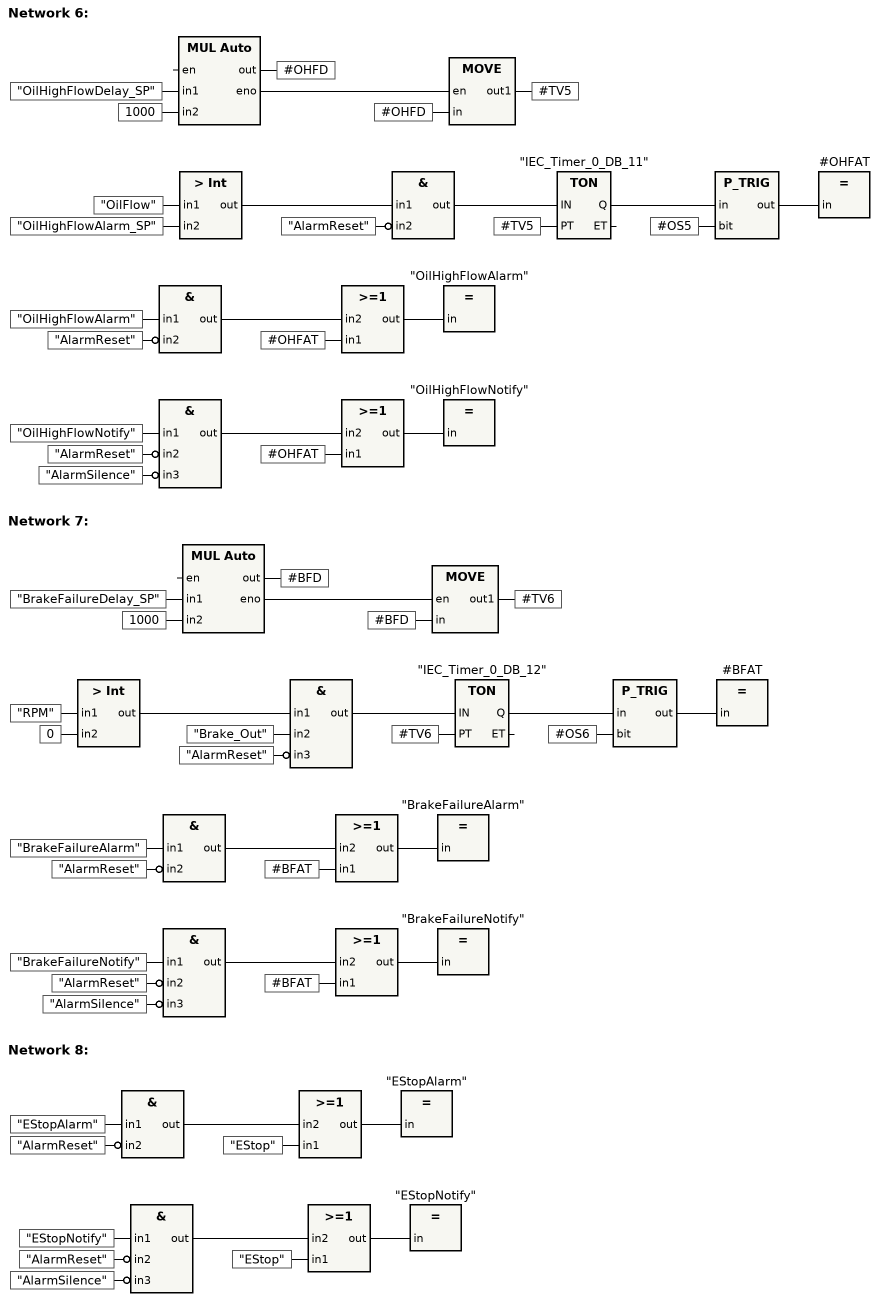
   #OHFD := "OilHighFlowDelay_SP" * 1000;
   #TV5 := #OHFD;
   "IEC_Timer_0_DB_11".TON(IN := ("OilFlow" > "OilHighFlowAlarm_SP") AND NOT "AlarmReset", PT := #TV5);
   #_w1 := "IEC_Timer_0_DB_11".Q AND NOT #OS5;   // rising edge
   #OS5 := "IEC_Timer_0_DB_11".Q;
   #OHFAT := #_w1;
   "OilHighFlowAlarm" := ("OilHighFlowAlarm" AND NOT "AlarmReset") OR #OHFAT;
   "OilHighFlowNotify" := ("OilHighFlowNotify" AND NOT "AlarmReset" AND NOT "AlarmSilence") OR #OHFAT;
END_REGION

REGION Network 7
   // Brake Failure Alarm
   #BFD := "BrakeFailureDelay_SP" * 1000;
   #TV6 := #BFD;
   "IEC_Timer_0_DB_12".TON(IN := ("RPM" > 0) AND "Brake_Out" AND NOT "AlarmReset", PT := #TV6);
   #_w1 := "IEC_Timer_0_DB_12".Q AND NOT #OS6;   // rising edge
   #OS6 := "IEC_Timer_0_DB_12".Q;
   #BFAT := #_w1;
   "BrakeFailureAlarm" := ("BrakeFailureAlarm" AND NOT "AlarmReset") OR #BFAT;
   "BrakeFailureNotify" := ("BrakeFailureNotify" AND NOT "AlarmReset" AND NOT "AlarmSilence") OR #BFAT;
END_REGION

REGION Network 8
   // E-Stop Alarm
   "EStopAlarm" := ("EStopAlarm" AND NOT "AlarmReset") OR "EStop";
   "EStopNotify" := ("EStopNotify" AND NOT "AlarmReset" AND NOT "AlarmSilence") OR "EStop";
END_REGION

REGION Network 9
   // Alarm Horn Control
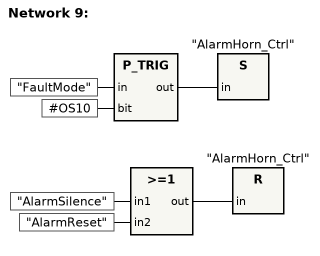
   #_w1 := "FaultMode" AND NOT #OS10;   // rising edge
   #OS10 := "FaultMode";
   IF #_w1 THEN "AlarmHorn_Ctrl" := TRUE; END_IF;
   IF "AlarmSilence" OR "AlarmReset" THEN "AlarmHorn_Ctrl" := FALSE; END_IF;
END_REGION
END_FUNCTION_BLOCK

FUNCTION_BLOCK "ALARMS_SCL"   // FB12, SCL
{ S7_Optimized_Access := 'TRUE' }
VERSION : 0.1
   VAR_TEMP
      OLFD : Int;
      TV1 : Time;
      OLFAT : Bool;
      T1 : Time;
      OCD : Int;
      TV2 : Time;
      OCAT : Bool;
      T2 : Time;
      HOTD : Int;
      TV3 : Time;
      HOTAT : Bool;
      T3 : Time;
      ROSD : Int;
      TV4 : Time;
      ROSAT : Bool;
      T4 : Time;
      OHFD : Int;
      TV5 : Time;
      OHFAT : Bool;
      T5 : Time;
      BFD : Int;
      TV6 : Time;
      BFAT : Bool;
      T6 : Time;
      ESAT : Bool;
   END_VAR
BEGIN
   // No P_TRIG to make these one-shots
   "AlarmReset" := "AlarmReset_PB";
   "AlarmSilence" := "AlarmSilence_PB";

   // Oil Low Flow Alarm
   #OLFD := "OilLowFlowDelay_SP" * 1000;
   "MOVE"(Int1:=#OLFD,
          Time1=>#TV1);

   IF "OilFlow" < "OilLowFlowAlarm_SP" AND "OilPumpVFDen_Out" AND NOT "Brake_Out" AND NOT "AlarmReset" THEN
       "IEC_Timer_0_DB_13".TON(IN := TRUE,
                               PT := #TV1,
                               Q => #OLFAT,
                               ET => #T1);
   ELSE
       RESET_TIMER("IEC_Timer_0_DB_13");
   END_IF;

   "OilLowFlowAlarm" := ("OilLowFlowAlarm" AND NOT "AlarmReset") OR #OLFAT;
   "OilLowFlowNotify" := ("OilLowFlowNotify" AND NOT "AlarmReset" AND NOT "AlarmSilence") OR #OLFAT;

   // Overcurrent Alarm
   #OCD := "OvercurrentDelay_SP" * 1000;
   "MOVE"(Int1 := #OCD,
          Time1 => #TV2);

   IF "Current" > "OvercurrentAlarm_SP" AND NOT "AlarmReset" THEN
       "IEC_Timer_0_DB_14".TON(IN := TRUE,
                               PT := #TV2,
                               Q => #OCAT,
                               ET => #T2);
   ELSE
       RESET_TIMER("IEC_Timer_0_DB_14");
   END_IF;

   "OvercurrentAlarm" := ("OvercurrentAlarm" AND NOT "AlarmReset") OR #OCAT;
   "OvercurrentNotify" := ("OvercurrentNotify" AND NOT "AlarmReset" AND NOT "AlarmSilence") OR #OCAT;

   // High Oil Temp Alarm
   #HOTD := "HighOilTempDelay_SP" * 1000;
   "MOVE"(Int1 := #HOTD,
          Time1 => #TV3);

   IF "OilTemp" > "HighOilTempAlarm_SP" AND NOT "AlarmReset" THEN
       "IEC_Timer_0_DB_15".TON(IN := TRUE,
                               PT := #TV3,
                               Q => #HOTAT,
                               ET => #T3);
   ELSE
       RESET_TIMER("IEC_Timer_0_DB_15");
   END_IF;

   "HighOilTempAlarm" := ("HighOilTempAlarm" AND NOT "AlarmReset") OR #HOTAT;
   "HighOilTempNotify" := ("HighOilTempNotify" AND NOT "AlarmReset" AND NOT "AlarmSilence") OR #HOTAT;

   // Rotor Overspeed Alarm
   #ROSD := "RotorOverspeedDelay_SP" * 1000;
   "MOVE"(Int1 := #ROSD,
          Time1 => #TV4);

   IF "RPM" > "RotorOverspeedAlarm_SP" AND NOT "AlarmReset" THEN
       "IEC_Timer_0_DB_16".TON(IN := TRUE,
                               PT := #TV4,
                               Q => #ROSAT,
                               ET => #T4);
   ELSE
       RESET_TIMER("IEC_Timer_0_DB_16");
   END_IF;

   "RotorOverspeedAlarm" := ("RotorOverspeedAlarm" AND NOT "AlarmReset") OR #ROSAT;
   "RotorOverspeedNotify" := ("RotorOverspeedNotify" AND NOT "AlarmReset" AND NOT "AlarmSilence") OR #ROSAT;

   // Oil High Flow Alarm
   #OHFD := "OilHighFlowDelay_SP" * 1000;
   "MOVE"(Int1 := #OHFD,
          Time1 => #TV5);

   IF "OilFlow" > "OilHighFlowAlarm_SP" AND NOT "AlarmReset" THEN
       "IEC_Timer_0_DB_17".TON(IN := TRUE,
                               PT := #TV5,
                               Q => #OHFAT,
                               ET => #T5);
   ELSE
       RESET_TIMER("IEC_Timer_0_DB_17");
   END_IF;

   "OilHighFlowAlarm" := ("OilHighFlowAlarm" AND NOT "AlarmReset") OR #OHFAT;
   "OilHighFlowNotify" := ("OilHighFlowNotify" AND NOT "AlarmReset" AND NOT "AlarmSilence") OR #OHFAT;

   // Brake Failure Alarm
   #BFD := "BrakeFailureDelay_SP" * 1000;
   "MOVE"(Int1 := #BFD,
          Time1 => #TV6);

   IF "RPM" > 0 AND "Brake_Out" AND NOT "AlarmReset" THEN
       "IEC_Timer_0_DB_18".TON(IN := TRUE,
                               PT := #TV6,
                               Q => #BFAT,
                               ET => #T6);
   ELSE
       RESET_TIMER("IEC_Timer_0_DB_18");
   END_IF;

   "BrakeFailureAlarm" := ("BrakeFailureAlarm" AND NOT "AlarmReset") OR #BFAT;
   "BrakeFailureNotify" := ("BrakeFailureNotify" AND NOT "AlarmReset" AND NOT "AlarmSilence") OR #BFAT;

   // E-Stop Alarm
   "EStopAlarm" := ("EStopAlarm" AND NOT "AlarmReset") OR "EStop";
   "EStopNotify" := ("EStopNotify" AND NOT "AlarmReset" AND NOT "AlarmSilence") OR "EStop";

   // Alarm Horn Control
   IF "FaultMode" AND NOT "AlarmHorn_Ctrl" THEN
       "AlarmHorn_Ctrl" := 1;
   END_IF;

   IF "AlarmHorn_Ctrl" AND ("AlarmReset" OR "AlarmSilence") THEN
       "AlarmHorn_Ctrl" := 0;
   END_IF;
END_FUNCTION_BLOCK

FUNCTION_BLOCK "ALARMS_STL"   // FB13, STL
{ S7_Optimized_Access := 'TRUE' }
VERSION : 0.1
   VAR
      OS1 : Bool;
      OS2 : Bool;
      OS3 : Bool;
      OS4 : Bool;
      OS5 : Bool;
      OS6 : Bool;
      OS7 : Bool;
      OS8 : Bool;
      OS9 : Bool;
      OS10 : Bool;
      OS11 : Bool;
      OS12 : Bool;
      OS13 : Bool;
      OS14 : Bool;
      OS15 : Bool;
      OS16 : Bool;
   END_VAR
   VAR_TEMP
      TV1 : Time;
      OLFAT : Bool;
      T1 : Time;
      TV2 : Time;
      OCAT : Bool;
      T2 : Time;
      TV3 : Time;
      HOTAT : Bool;
      T3 : Time;
      TV4 : Time;
      ROSAT : Bool;
      T4 : Time;
      TV5 : Time;
      OHFAT : Bool;
      T5 : Time;
      TV6 : Time;
      BFAT : Bool;
      T6 : Time;
      ESAT : Bool;
   END_VAR
BEGIN

REGION Network 1
   AlarmReset_PB:A     "AlarmReset_PB";
         JC    SetAlarmReset;
         JU    ResetAlarmReset;

   SetAlarmReset:SET;
         S     "AlarmReset";
         JU    AlarmSilence_PB;

   ResetAlarmReset:R     "AlarmReset";
         JU    AlarmSilence_PB;

   AlarmSilence_PB:A     "AlarmSilence_PB";
         JC    SetAlarmSilence;
         JU    ResetAlarmSilence;

   SetAlarmSilence:SET;
         S     "AlarmSilence";
         JU    OilLowFlowAlarm;

   ResetAlarmSilence:R     "AlarmSilence";
         JU    OilLowFlowAlarm;
END_REGION

REGION Network 2
   // Oil Low Flow Alarm
   OilLowFlowAlarm:A     "AlarmReset";
         FP    #OS1;
         JC    ResetOLFAlarm;
         CLR;
         A     "AlarmSilence";
         FP    #OS2;
         JC    ResetOLFNotify;
         CLR;
         L     "OilFlow";
         L     "OilLowFlowAlarm_SP";
         <I;
         A     "OilPumpVFDen_Out";
         AN    "Brake_Out";
         JC    OLFTimer;
         JU    OvercurrentAlarm;

   OLFTimer:CALL  "MOVE"
         ( Int1  := "OilLowFlowDelay_SP",
           Time1 := #TV1
         );
         CALL  TON, "IEC_Timer_0_DB_19"
         ( IN := TRUE,
           PT := #TV1,
           Q  := #OLFAT,
           ET := #T1
         );
         A     #OLFAT;
         JC    SetOLFAlarm;
         JU    OvercurrentAlarm;

   SetOLFAlarm:SET;
         S     "OilLowFlowAlarm";
         S     "OilLowFlowNotify";
         JU    OvercurrentAlarm;

   ResetOLFAlarm:R     "OilLowFlowAlarm";
         R     "OilLowFlowNotify";
         CALL  RESET_TIMER
         ( "TIMER" := "IEC_Timer_0_DB_19"
         );
         JU    OvercurrentAlarm;

   ResetOLFNotify:R     "OilLowFlowNotify";
         JU    OvercurrentAlarm;
END_REGION

REGION Network 3
   // Overcurrent Alarm
   OvercurrentAlarm:A     "AlarmReset";
         FP    #OS3;
         JC    ResetOCAlarm;
         CLR;
         A     "AlarmSilence";
         FP    #OS4;
         JC    ResetOCNotify;
         CLR;
         L     "Current";
         L     "OvercurrentAlarm_SP";
         >I;
         JC    OCTimer;
         JU    HighOilTempAlarm;

   OCTimer:CALL  "MOVE"
         ( Int1  := "OvercurrentDelay_SP",
           Time1 := #TV2
         );
         CALL  TON, "IEC_Timer_0_DB_20"
         ( IN := TRUE,
           PT := #TV2,
           Q  := #OCAT,
           ET := #T2
         );
         A     #OCAT;
         JC    SetOCAlarm;
         JU    HighOilTempAlarm;

   SetOCAlarm:SET;
         S     "OvercurrentAlarm";
         S     "OvercurrentNotify";
         JU    HighOilTempAlarm;

   ResetOCAlarm:R     "OvercurrentAlarm";
         R     "OvercurrentNotify";
         CALL  RESET_TIMER
         ( "TIMER" := "IEC_Timer_0_DB_20"
         );
         JU    HighOilTempAlarm;

   ResetOCNotify:R     "OvercurrentNotify";
         JU    HighOilTempAlarm;
END_REGION

REGION Network 4
   // High Oil Temp Alarm
   HighOilTempAlarm:A     "AlarmReset";
         FP    #OS5;
         JC    ResetHOTAlarm;
         CLR;
         A     "AlarmSilence";
         FP    #OS6;
         JC    ResetHOTNotify;
         CLR;
         L     "OilTemp";
         L     "HighOilTempAlarm_SP";
         >I;
         JC    HOTTimer;
         JU    RotorOverspeedAlarm;

   HOTTimer:CALL  "MOVE"
         ( Int1  := "HighOilTempDelay_SP",
           Time1 := #TV3
         );
         CALL  TON, "IEC_Timer_0_DB_21"
         ( IN := TRUE,
           PT := #TV3,
           Q  := #HOTAT,
           ET := #T3
         );
         A     #HOTAT;
         JC    SetHOTAlarm;
         JU    RotorOverspeedAlarm;

   SetHOTAlarm:SET;
         S     "HighOilTempAlarm";
         S     "HighOilTempNotify";
         JU    RotorOverspeedAlarm;

   ResetHOTAlarm:R     "HighOilTempAlarm";
         R     "HighOilTempNotify";
         CALL  RESET_TIMER
         ( "TIMER" := "IEC_Timer_0_DB_21"
         );
         JU    RotorOverspeedAlarm;

   ResetHOTNotify:R     "HighOilTempNotify";
         JU    RotorOverspeedAlarm;
END_REGION

REGION Network 5
   // Rotor Overspeed Alarm
   RotorOverspeedAlarm:A     "AlarmReset";
         FP    #OS7;
         JC    ResetROSAlarm;
         CLR;
         A     "AlarmSilence";
         FP    #OS8;
         JC    ResetROSNotify;
         CLR;
         L     "RPM";
         L     "RotorOverspeedAlarm_SP";
         >I;
         JC    ROSTimer;
         JU    OilHighFlowAlarm;

   ROSTimer:CALL  "MOVE"
         ( Int1  := "RotorOverspeedDelay_SP",
           Time1 := #TV4
         );
         CALL  TON, "IEC_Timer_0_DB_22"
         ( IN := TRUE,
           PT := #TV4,
           Q  := #ROSAT,
           ET := #T4
         );
         A     #ROSAT;
         JC    SetROSAlarm;
         JU    OilHighFlowAlarm;

   SetROSAlarm:SET;
         S     "RotorOverspeedAlarm";
         S     "RotorOverspeedNotify";
         JU    OilHighFlowAlarm;

   ResetROSAlarm:R     "RotorOverspeedAlarm";
         R     "RotorOverspeedNotify";
         CALL  RESET_TIMER
         ( "TIMER" := "IEC_Timer_0_DB_22"
         );
         JU    OilHighFlowAlarm;

   ResetROSNotify:R     "RotorOverspeedNotify";
         JU    OilHighFlowAlarm;
END_REGION

REGION Network 6
   // Oil High Flow Alarm
   OilHighFlowAlarm:A     "AlarmReset";
         FP    #OS9;
         JC    ResetOHFAlarm;
         CLR;
         A     "AlarmSilence";
         FP    #OS10;
         JC    ResetOHFNotify;
         CLR;
         L     "OilFlow";
         L     "OilHighFlowAlarm_SP";
         >I;
         JC    OHFTimer;
         JU    BrakeFailureAlarm;

   OHFTimer:CALL  "MOVE"
         ( Int1  := "OilHighFlowDelay_SP",
           Time1 := #TV5
         );
         CALL  TON, "IEC_Timer_0_DB_23"
         ( IN := TRUE,
           PT := #TV5,
           Q  := #OHFAT,
           ET := #T5
         );
         A     #OHFAT;
         JC    SetOHFAlarm;
         JU    BrakeFailureAlarm;

   SetOHFAlarm:SET;
         S     "OilHighFlowAlarm";
         S     "OilHighFlowNotify";
         JU    BrakeFailureAlarm;

   ResetOHFAlarm:R     "OilHighFlowAlarm";
         R     "OilHighFlowNotify";
         CALL  RESET_TIMER
         ( "TIMER" := "IEC_Timer_0_DB_23"
         );
         JU    BrakeFailureAlarm;

   ResetOHFNotify:R     "OilHighFlowNotify";
         JU    BrakeFailureAlarm;
END_REGION

REGION Network 7
   // Brake Failure Alarm
   BrakeFailureAlarm:A     "AlarmReset";
         FP    #OS11;
         JC    ResetBFAlarm;
         CLR;
         A     "AlarmSilence";
         FP    #OS12;
         JC    ResetBFNotify;
         CLR;
         L     "RPM";
         L     0;
         >I;
         A     "Brake_Out";
         JC    BFTimer;
         JU    EStopAlarm;

   BFTimer:CALL  "MOVE"
         ( Int1  := "BrakeFailureDelay_SP",
           Time1 := #TV6
         );
         CALL  TON, "IEC_Timer_0_DB_24"
         ( IN := TRUE,
           PT := #TV6,
           Q  := #BFAT,
           ET := #T6
         );
         A     #BFAT;
         JC    SetBFAlarm;
         JU    EStopAlarm;

   SetBFAlarm:SET;
         S     "BrakeFailureAlarm";
         S     "BrakeFailureNotify";
         JU    EStopAlarm;

   ResetBFAlarm:R     "BrakeFailureAlarm";
         R     "BrakeFailureNotify";
         CALL  RESET_TIMER
         ( "TIMER" := "IEC_Timer_0_DB_24"
         );
         JU    EStopAlarm;

   ResetBFNotify:R     "BrakeFailureNotify";
         JU    EStopAlarm;
END_REGION

REGION Network 8
   // E-Stop Alarm
   EStopAlarm:A     "AlarmReset";
         FP    #OS13;
         JC    ResetESAlarm;
         CLR;
         A     "AlarmSilence";
         FP    #OS14;
         JC    ResetESNotify;
         CLR;
         A     "EStop";
         JC    SetESAlarm;
         JU    AlarmHornControl;

   SetESAlarm:SET;
         S     "EStopAlarm";
         S     "EStopNotify";
         JU    AlarmHornControl;

   ResetESAlarm:R     "EStopAlarm";
         R     "EStopNotify";
         JU    AlarmHornControl;

   ResetESNotify:R     "EStopNotify";
         JU    AlarmHornControl;
END_REGION

REGION Network 9
   // Alarm Horn Control
   AlarmHornControl:A     "FaultMode";
         FP    #OS15;
         JC    SetAlarmHorn;
         CLR;
         A     "AlarmReset";
         O     "AlarmSilence";
         FP    #OS16;
         JC    ResetAlarmHorn;
         JU    EndOfLine;

   SetAlarmHorn:SET;
         S     "AlarmHorn_Ctrl";
         JU    EndOfLine;

   ResetAlarmHorn:R     "AlarmHorn_Ctrl";
         JU    EndOfLine;

   EndOfLine:BE;
END_REGION
END_FUNCTION_BLOCK

FUNCTION_BLOCK "MODES_LAD"   // FB14, LAD
{ S7_Optimized_Access := 'TRUE' }
VERSION : 0.1
   VAR
      OS1 : Bool;
      OS2 : Bool;
      OS3 : Bool;
      OS4 : Bool;
      OS5 : Bool;
   END_VAR
   VAR_TEMP
      TV1 : Time;
      WMD : Int;
      StabilizekW_Min : Int;
      StabilizekW_Max : Int;
      SMD : Int;
      TV2 : Time;
      CMD : Int;
      TV3 : Time;
   END_VAR
   VAR_TEMP   // added for the SCL form of the ladder/FBD networks
      _w1 : Bool;
      _w2 : Bool;
      _w3 : Bool;
   END_VAR
BEGIN

REGION Network 1: Warmup Mode
   // When Start pushbutton is pressed, the sequence begins with this step. Allow the rotor to turn at a speed somewhere between 20 and 50 RPMs and run the oil pump at some low output level (2-10 GPM maybe?) until the oil temp reaches 150 degrees. Once we’ve maintained at least 150 degrees for 10 seconds, we want to transition into the next mode.
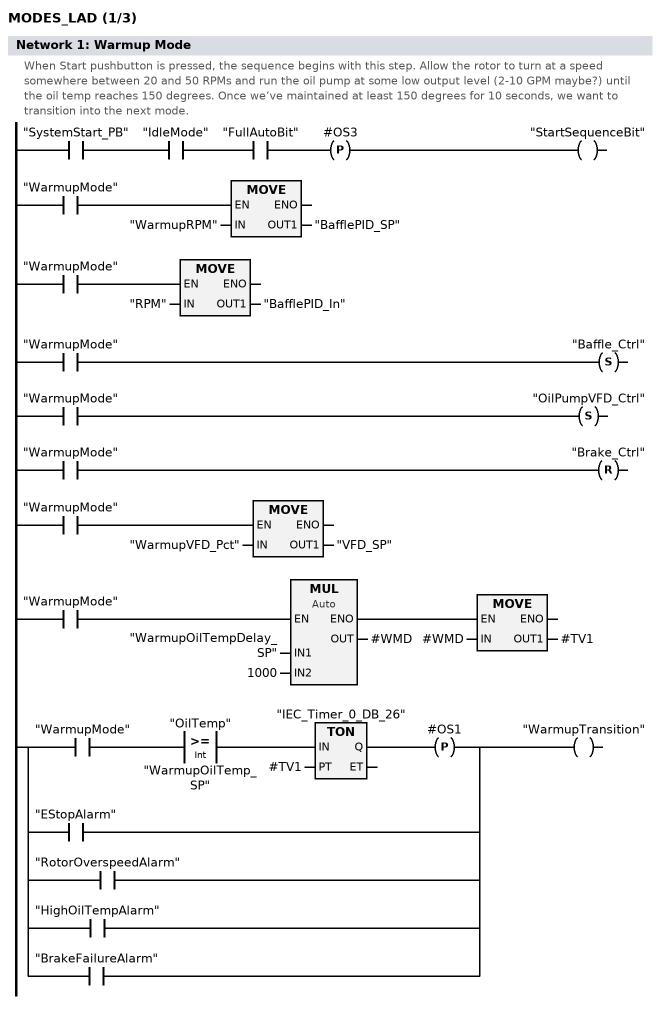
   #_w1 := "SystemStart_PB" AND "IdleMode" AND "FullAutoBit";
   #_w2 := #_w1 AND NOT #OS3;   // rising edge
   #OS3 := #_w1;
   "StartSequenceBit" := #_w2;
   IF "WarmupMode" THEN
       "BafflePID_SP" := "WarmupRPM";
       "BafflePID_In" := "RPM";
       "Baffle_Ctrl" := TRUE;
       "OilPumpVFD_Ctrl" := TRUE;
       "Brake_Ctrl" := FALSE;
       "VFD_SP" := "WarmupVFD_Pct";
       #WMD := "WarmupOilTempDelay_SP" * 1000;
       #TV1 := #WMD;
   END_IF;
   "IEC_Timer_0_DB_26".TON(IN := "WarmupMode" AND ("OilTemp" >= "WarmupOilTemp_SP"), PT := #TV1);
   #_w3 := "IEC_Timer_0_DB_26".Q AND NOT #OS1;   // rising edge
   #OS1 := "IEC_Timer_0_DB_26".Q;
   "WarmupTransition" := #_w3 OR "EStopAlarm" OR "RotorOverspeedAlarm" OR "HighOilTempAlarm" OR "BrakeFailureAlarm";
END_REGION

REGION Network 2: Stabilize Mode
   // Generator should speed up until desired kW output is attained. Once we’re stable within 5kW (+/-) of the setpoint for at least 10 seconds, we should transition into the next mode.
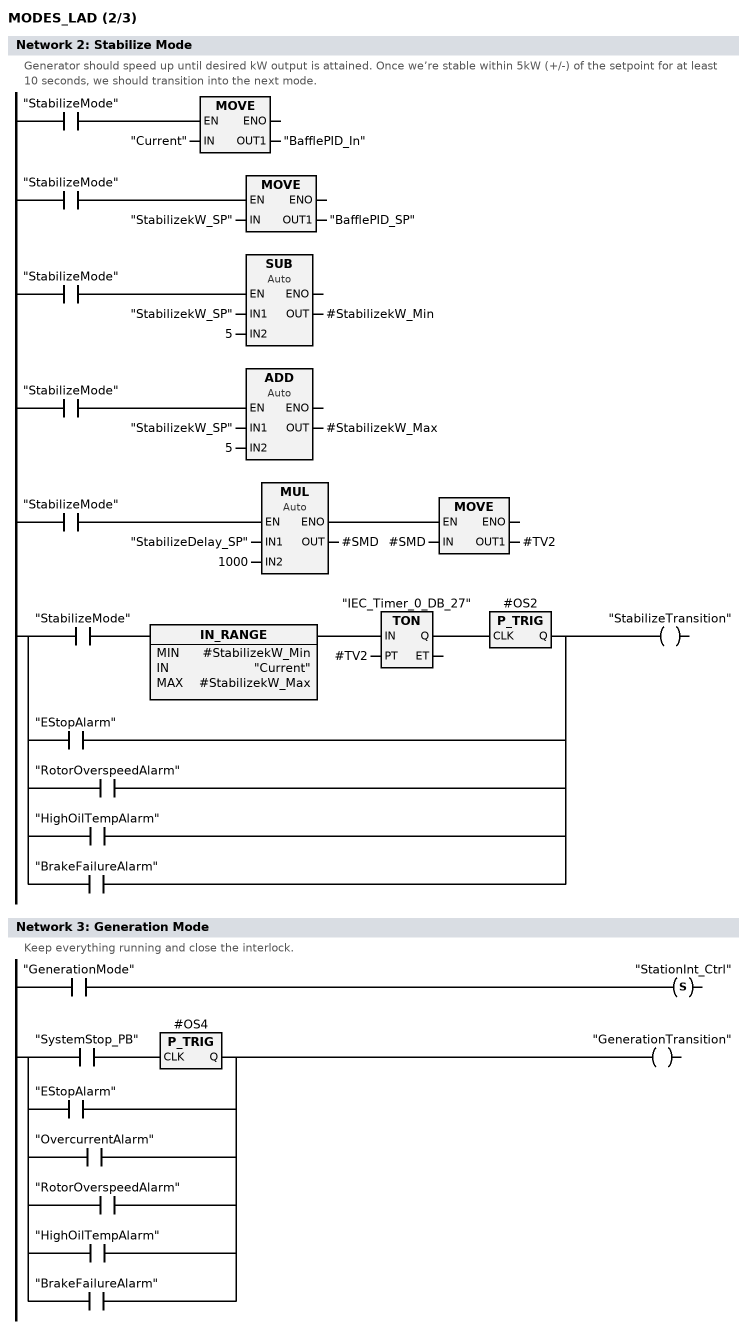
   IF "StabilizeMode" THEN
       "BafflePID_In" := "Current";
       "BafflePID_SP" := "StabilizekW_SP";
       #StabilizekW_Min := "StabilizekW_SP" - 5;
       #StabilizekW_Max := "StabilizekW_SP" + 5;
       #SMD := "StabilizeDelay_SP" * 1000;
       #TV2 := #SMD;
   END_IF;
   "IEC_Timer_0_DB_27".TON(IN := "StabilizeMode" AND (#StabilizekW_Min <= "Current") AND ("Current" <= #StabilizekW_Max),
                           PT := #TV2);
   #_w1 := "IEC_Timer_0_DB_27".Q AND NOT #OS2;   // rising edge
   #OS2 := "IEC_Timer_0_DB_27".Q;
   "StabilizeTransition" := #_w1 OR "EStopAlarm" OR "RotorOverspeedAlarm" OR "HighOilTempAlarm" OR "BrakeFailureAlarm";
END_REGION

REGION Network 3: Generation Mode
   // Keep everything running and close the interlock.
   RUNG wire#powerrail
      Contact( "GenerationMode" )
      S_Coil( "StationInt_Ctrl" )
   END_RUNG
   RUNG wire#powerrail
      Contact( "SystemStop_PB" )
      P_Trig( #OS4 )
      wire#w1
      Coil( "GenerationTransition" )
   END_RUNG
   RUNG wire#powerrail
      Contact( "EStopAlarm" )
   END_RUNG wire#w1
   RUNG wire#powerrail
      Contact( "OvercurrentAlarm" )
   END_RUNG wire#w1
   RUNG wire#powerrail
      Contact( "RotorOverspeedAlarm" )
   END_RUNG wire#w1
   RUNG wire#powerrail
      Contact( "HighOilTempAlarm" )
   END_RUNG wire#w1
   RUNG wire#powerrail
      Contact( "BrakeFailureAlarm" )
   END_RUNG wire#w1
   // the same network as SCL:
   IF "GenerationMode" THEN "StationInt_Ctrl" := TRUE; END_IF;
   #_w1 := "SystemStop_PB" AND NOT #OS4;   // rising edge
   #OS4 := "SystemStop_PB";
   "GenerationTransition" := #_w1 OR "EStopAlarm" OR "OvercurrentAlarm" OR "RotorOverspeedAlarm" OR "HighOilTempAlarm" OR "BrakeFailureAlarm";
END_REGION

REGION Network 4: Cooldown Mode
   // Once the Stop button has been pushed, open the interlock, slow the rotor to between 20 and 50 RPMs and maintain a high oil flow until the oil temp is below 150 degrees. Once we’re below for ten seconds, we transition into Idle mode.
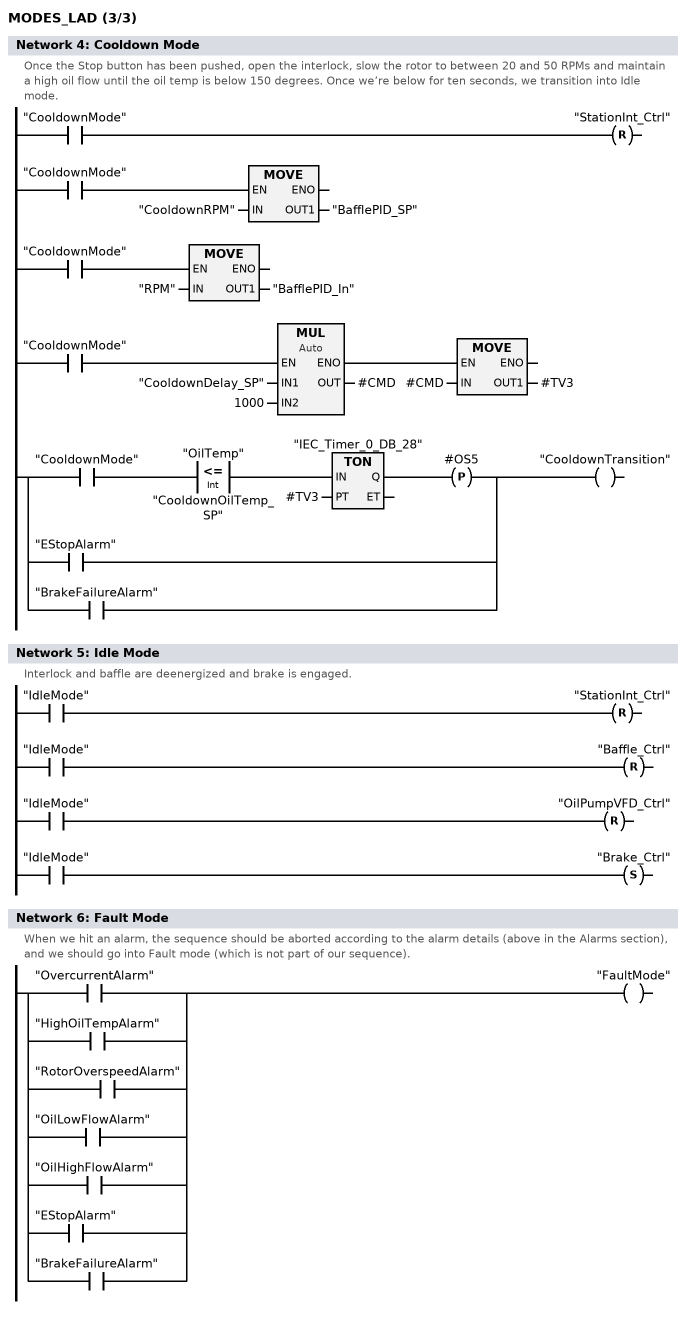
   IF "CooldownMode" THEN
       "StationInt_Ctrl" := FALSE;
       "BafflePID_SP" := "CooldownRPM";
       "BafflePID_In" := "RPM";
       #CMD := "CooldownDelay_SP" * 1000;
       #TV3 := #CMD;
   END_IF;
   "IEC_Timer_0_DB_28".TON(IN := "CooldownMode" AND ("OilTemp" <= "CooldownOilTemp_SP"), PT := #TV3);
   #_w1 := "IEC_Timer_0_DB_28".Q AND NOT #OS5;   // rising edge
   #OS5 := "IEC_Timer_0_DB_28".Q;
   "CooldownTransition" := #_w1 OR "EStopAlarm" OR "BrakeFailureAlarm";
END_REGION

REGION Network 5: Idle Mode
   // Interlock and baffle are deenergized and brake is engaged.
   RUNG wire#powerrail
      Contact( "IdleMode" )
      R_Coil( "StationInt_Ctrl" )
   END_RUNG
   RUNG wire#powerrail
      Contact( "IdleMode" )
      R_Coil( "Baffle_Ctrl" )
   END_RUNG
   RUNG wire#powerrail
      Contact( "IdleMode" )
      R_Coil( "OilPumpVFD_Ctrl" )
   END_RUNG
   RUNG wire#powerrail
      Contact( "IdleMode" )
      S_Coil( "Brake_Ctrl" )
   END_RUNG
   // the same network as SCL:
   IF "IdleMode" THEN
       "StationInt_Ctrl" := FALSE;
       "Baffle_Ctrl" := FALSE;
       "OilPumpVFD_Ctrl" := FALSE;
       "Brake_Ctrl" := TRUE;
   END_IF;
END_REGION

REGION Network 6: Fault Mode
   // When we hit an alarm, the sequence should be aborted according to the alarm details (above in the Alarms section), and we should go into Fault mode (which is not part of our sequence).
   RUNG wire#powerrail
      Contact( "OvercurrentAlarm" )
      wire#w1
      Coil( "FaultMode" )
   END_RUNG
   RUNG wire#powerrail
      Contact( "HighOilTempAlarm" )
   END_RUNG wire#w1
   RUNG wire#powerrail
      Contact( "RotorOverspeedAlarm" )
   END_RUNG wire#w1
   RUNG wire#powerrail
      Contact( "OilLowFlowAlarm" )
   END_RUNG wire#w1
   RUNG wire#powerrail
      Contact( "OilHighFlowAlarm" )
   END_RUNG wire#w1
   RUNG wire#powerrail
      Contact( "EStopAlarm" )
   END_RUNG wire#w1
   RUNG wire#powerrail
      Contact( "BrakeFailureAlarm" )
   END_RUNG wire#w1
   // the same network as SCL:
   "FaultMode" := "OvercurrentAlarm" OR "HighOilTempAlarm" OR "RotorOverspeedAlarm" OR "OilLowFlowAlarm" OR "OilHighFlowAlarm" OR "EStopAlarm" OR "BrakeFailureAlarm";
END_REGION
END_FUNCTION_BLOCK

FUNCTION_BLOCK "MODES_FBD"   // FB15, FBD
{ S7_Optimized_Access := 'TRUE' }
VERSION : 0.1
   VAR
      OS1 : Bool;
      OS2 : Bool;
      OS3 : Bool;
      OS4 : Bool;
      OS5 : Bool;
   END_VAR
   VAR_TEMP
      WMD : Int;
      TV1 : Time;
      StabilizekW_Min : Int;
      StabilizekW_Max : Int;
      SMD : Int;
      TV2 : Time;
      CMD : Int;
      TV3 : Time;
   END_VAR
   VAR_TEMP   // added for the SCL form of the ladder/FBD networks
      _w1 : Bool;
      _w2 : Bool;
      _w3 : Bool;
   END_VAR
BEGIN

REGION Network 1: Warmup Mode
   // When Start pushbutton is pressed, the sequence begins with this step. Allow the rotor to turn at a speed somewhere between 20 and 50 RPMs and run the oil pump at some low output level (2-10 GPM maybe?) until the oil temp reaches 150 degrees. Once we’ve maintained at least 150 degrees for 10 seconds, we want to transition into the next mode.
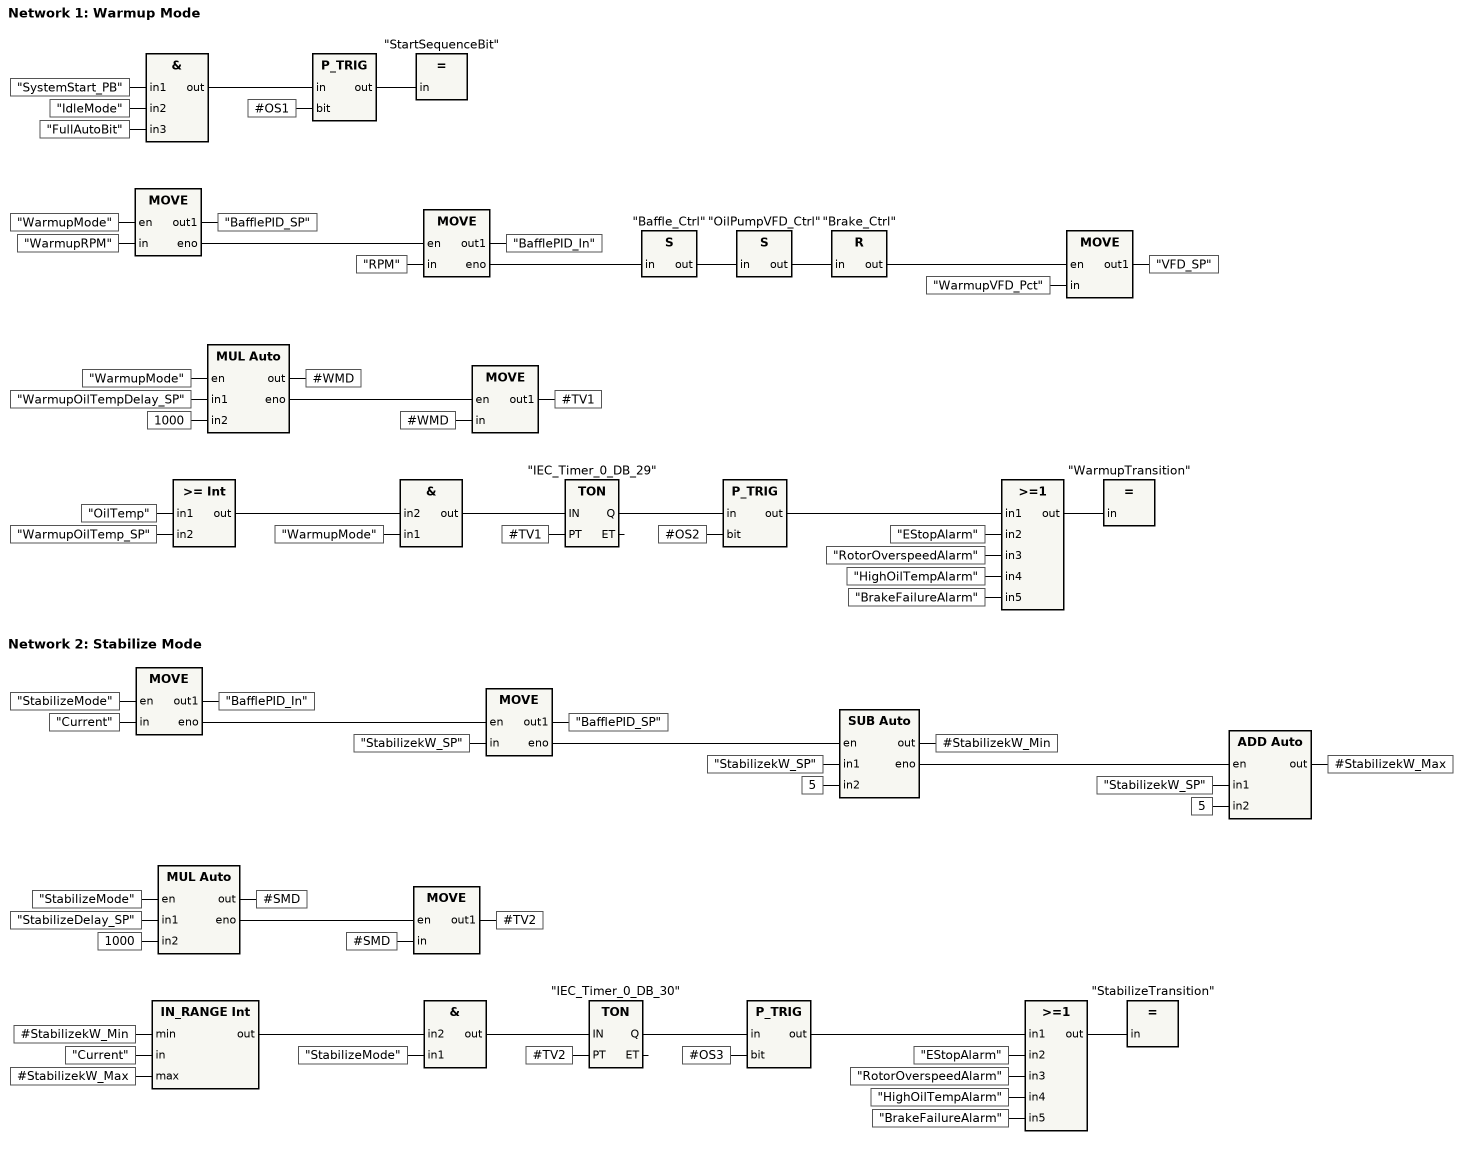
   #_w1 := "SystemStart_PB" AND "IdleMode" AND "FullAutoBit";
   #_w2 := #_w1 AND NOT #OS1;   // rising edge
   #OS1 := #_w1;
   "StartSequenceBit" := #_w2;
   IF "WarmupMode" THEN
       "BafflePID_SP" := "WarmupRPM";
       "BafflePID_In" := "RPM";
       "Baffle_Ctrl" := TRUE;
       "OilPumpVFD_Ctrl" := TRUE;
       "Brake_Ctrl" := FALSE;
       "VFD_SP" := "WarmupVFD_Pct";
       #WMD := "WarmupOilTempDelay_SP" * 1000;
       #TV1 := #WMD;
   END_IF;
   "IEC_Timer_0_DB_29".TON(IN := ("OilTemp" >= "WarmupOilTemp_SP") AND "WarmupMode", PT := #TV1);
   #_w3 := "IEC_Timer_0_DB_29".Q AND NOT #OS2;   // rising edge
   #OS2 := "IEC_Timer_0_DB_29".Q;
   "WarmupTransition" := #_w3 OR "EStopAlarm" OR "RotorOverspeedAlarm" OR "HighOilTempAlarm" OR "BrakeFailureAlarm";
END_REGION

REGION Network 2: Stabilize Mode
   // Generator should speed up until desired kW output is attained. Once we’re stable within 5kW (+/-) of the setpoint for at least 10 seconds, we should transition into the next mode.
   IF "StabilizeMode" THEN
       "BafflePID_In" := "Current";
       "BafflePID_SP" := "StabilizekW_SP";
       #StabilizekW_Min := "StabilizekW_SP" - 5;
       #StabilizekW_Max := "StabilizekW_SP" + 5;
       #SMD := "StabilizeDelay_SP" * 1000;
       #TV2 := #SMD;
   END_IF;
   "IEC_Timer_0_DB_30".TON(IN := (#StabilizekW_Min <= "Current") AND ("Current" <= #StabilizekW_Max) AND "StabilizeMode",
                           PT := #TV2);
   #_w1 := "IEC_Timer_0_DB_30".Q AND NOT #OS3;   // rising edge
   #OS3 := "IEC_Timer_0_DB_30".Q;
   "StabilizeTransition" := #_w1 OR "EStopAlarm" OR "RotorOverspeedAlarm" OR "HighOilTempAlarm" OR "BrakeFailureAlarm";
END_REGION

REGION Network 3: Generation Mode
   // Keep everything running and close the interlock.
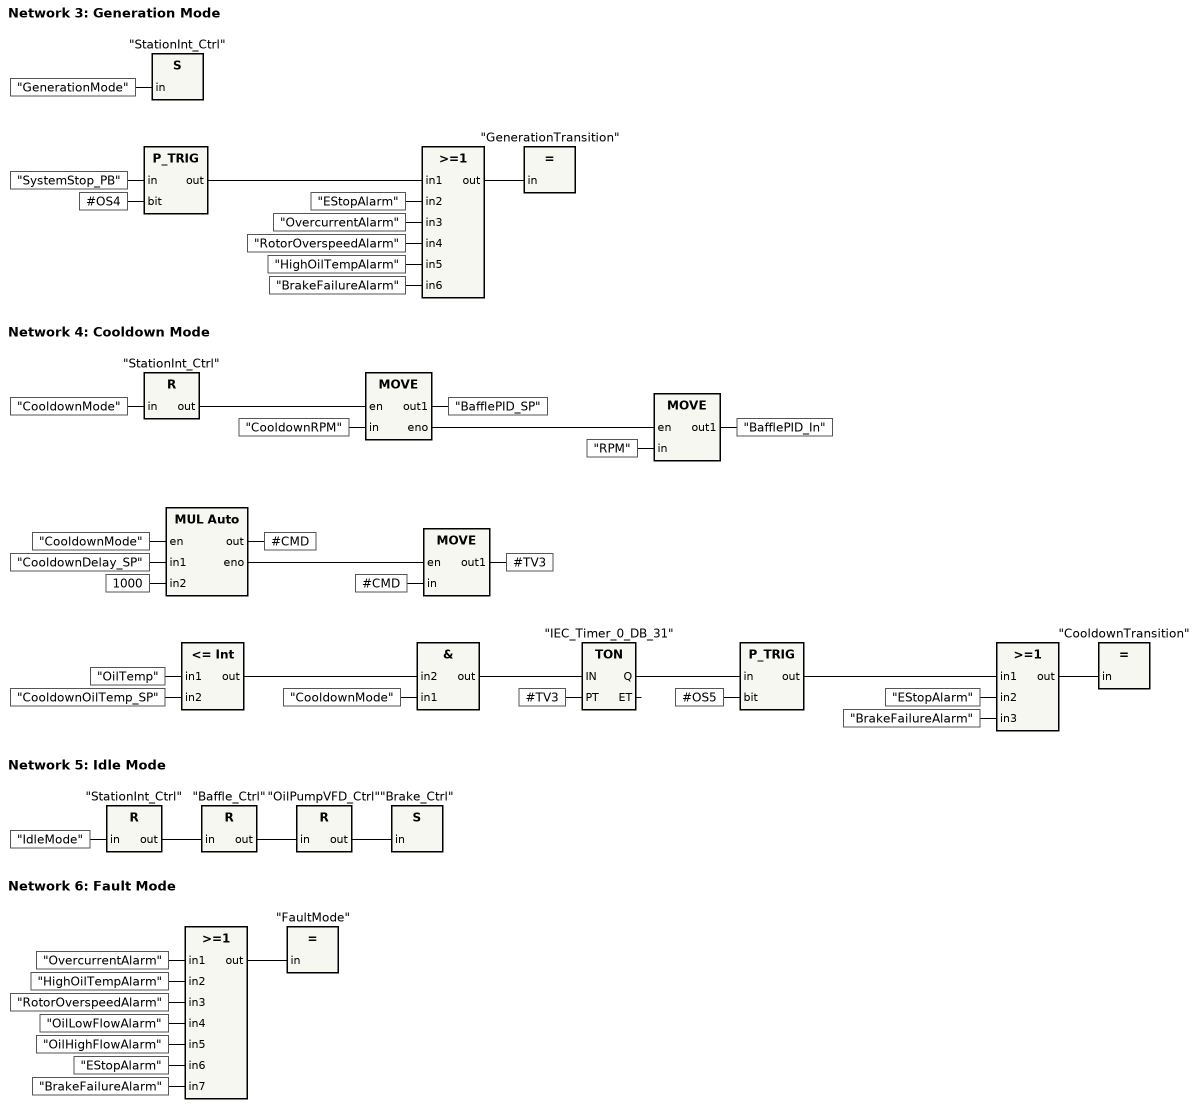
   IF "GenerationMode" THEN "StationInt_Ctrl" := TRUE; END_IF;
   #_w1 := "SystemStop_PB" AND NOT #OS4;   // rising edge
   #OS4 := "SystemStop_PB";
   "GenerationTransition" := #_w1 OR "EStopAlarm" OR "OvercurrentAlarm" OR "RotorOverspeedAlarm" OR "HighOilTempAlarm" OR "BrakeFailureAlarm";
END_REGION

REGION Network 4: Cooldown Mode
   // Once the Stop button has been pushed, open the interlock, slow the rotor to between 20 and 50 RPMs and maintain a high oil flow until the oil temp is below 150 degrees. Once we’re below for ten seconds, we transition into Idle mode.
   IF "CooldownMode" THEN
       "StationInt_Ctrl" := FALSE;
       "BafflePID_SP" := "CooldownRPM";
       "BafflePID_In" := "RPM";
       #CMD := "CooldownDelay_SP" * 1000;
       #TV3 := #CMD;
   END_IF;
   "IEC_Timer_0_DB_31".TON(IN := ("OilTemp" <= "CooldownOilTemp_SP") AND "CooldownMode", PT := #TV3);
   #_w1 := "IEC_Timer_0_DB_31".Q AND NOT #OS5;   // rising edge
   #OS5 := "IEC_Timer_0_DB_31".Q;
   "CooldownTransition" := #_w1 OR "EStopAlarm" OR "BrakeFailureAlarm";
END_REGION

REGION Network 5: Idle Mode
   // Interlock and baffle are deenergized and brake is engaged.
   IF "IdleMode" THEN
       "StationInt_Ctrl" := FALSE;
       "Baffle_Ctrl" := FALSE;
       "OilPumpVFD_Ctrl" := FALSE;
       "Brake_Ctrl" := TRUE;
   END_IF;
END_REGION

REGION Network 6: Fault Mode
   // When we hit an alarm, the sequence should be aborted according to the alarm details (above in the Alarms section), and we should go into Fault mode (which is not part of our sequence).
   "FaultMode" := "OvercurrentAlarm" OR "HighOilTempAlarm" OR "RotorOverspeedAlarm" OR "OilLowFlowAlarm" OR "OilHighFlowAlarm" OR "EStopAlarm" OR "BrakeFailureAlarm";
END_REGION
END_FUNCTION_BLOCK

FUNCTION_BLOCK "MODES_SCL"   // FB16, SCL
{ S7_Optimized_Access := 'TRUE' }
VERSION : 0.1
   VAR_TEMP
      TV1 : Time;
      T1 : Time;
      WMT : Bool;
      StabilizekW_Min : Int;
      StabilizekW_Max : Int;
      TV2 : Time;
      SMT : Bool;
      T2 : Time;
      TV3 : Time;
      CMT : Bool;
      T3 : Time;
   END_VAR
BEGIN
   IF "EStopAlarm" OR "BrakeFailureAlarm" THEN
       "WarmupTransition" := TRUE;
       "StabilizeTransition" := TRUE;
       "GenerationTransition" := TRUE;
       "CooldownTransition" := TRUE;
   END_IF;

   IF "RotorOverspeedAlarm" OR "HighOilTempAlarm" THEN
       "WarmupTransition" := TRUE;
       "StabilizeTransition" := TRUE;
       "GenerationTransition" := TRUE;
   END_IF;

   // Warmup Mode
   IF "SystemStart_PB" AND "IdleMode" AND "FullAutoBit" THEN
       "StartSequenceBit" := TRUE;
   ELSE
       "StartSequenceBit" := FALSE;
   END_IF;

   IF "WarmupMode" THEN
       "BafflePID_SP" := "WarmupRPM";
       "BafflePID_In" := "RPM";
       "Baffle_Ctrl" := TRUE;
       "OilPumpVFD_Ctrl" := TRUE;
       "Brake_Ctrl" := FALSE;
       "VFD_SP" := "WarmupVFD_Pct";
       IF "OilTemp" >= "WarmupOilTemp_SP" THEN
           "MOVE"(Int1 := "WarmupOilTempDelay_SP",
                  Time1 => #TV1);
           "IEC_Timer_0_DB_32".TON(IN := TRUE,
                                   PT := #TV1,
                                   Q => #WMT,
                                   ET => #T1);
       ELSE
           RESET_TIMER("IEC_Timer_0_DB_32");
       END_IF;
       IF #WMT THEN
           RESET_TIMER("IEC_Timer_0_DB_32");
           "WarmupTransition" := TRUE;
       END_IF;
   ELSE
       "WarmupTransition" := FALSE;
   END_IF;

   // Stabilize Mode
   IF "StabilizeMode" THEN
       "BafflePID_In" := "Current";
       "BafflePID_SP" := "StabilizekW_SP";
       #StabilizekW_Min := "StabilizekW_SP" - 5;
       #StabilizekW_Max := "StabilizekW_SP" + 5;
       IF "Current" >= #StabilizekW_Min AND "Current" <= #StabilizekW_Max THEN
           "MOVE"(Int1 := "StabilizeDelay_SP",
                  Time1 => #TV2);
           "IEC_Timer_0_DB_33".TON(IN := TRUE,
                                   PT := #TV2,
                                   Q => #SMT,
                                   ET => #T2);
       ELSE
           RESET_TIMER("IEC_Timer_0_DB_33");
       END_IF;
       IF #SMT THEN
           RESET_TIMER("IEC_Timer_0_DB_33");
           "StabilizeTransition" := TRUE;
       END_IF;
   ELSE
       "StabilizeTransition" := FALSE;
   END_IF;

   // Generation Mode
   IF "GenerationMode" THEN
       "StationInt_Ctrl" := TRUE;
       IF "SystemStop_PB" OR "OvercurrentAlarm" THEN
           "GenerationTransition" := TRUE;
       END_IF;
   ELSE
       "GenerationTransition" := FALSE;
   END_IF;

   // Cooldown Mode
   IF "CooldownMode" THEN
       "StationInt_Ctrl" := FALSE;
       "BafflePID_SP" := "CooldownRPM";
       "BafflePID_In" := "RPM";
       IF "OilTemp" <= "CooldownOilTemp_SP" THEN
           "MOVE"(Int1 := "CooldownDelay_SP",
                  Time1 => #TV3);
           "IEC_Timer_0_DB_34".TON(IN := TRUE,
                                   PT := #TV3,
                                   Q => #CMT,
                                   ET => #T3);
       ELSE
           RESET_TIMER("IEC_Timer_0_DB_34");
       END_IF;
       IF #CMT THEN
           RESET_TIMER("IEC_Timer_0_DB_34");
           "CooldownTransition" := TRUE;
       END_IF;
   ELSE
       "CooldownTransition" := FALSE;
   END_IF;

   // Idle Mode
   IF "IdleMode" THEN
       "StationInt_Ctrl" := FALSE;
       "Baffle_Ctrl" := FALSE;
       "OilPumpVFD_Ctrl" := FALSE;
       "Brake_Ctrl" := TRUE;
   END_IF;

   // Fault Mode
   IF "OvercurrentAlarm" OR "HighOilTempAlarm" OR "RotorOverspeedAlarm" OR "OilLowFlowAlarm" OR "OilHighFlowAlarm" OR "EStopAlarm" OR "BrakeFailureAlarm" THEN
       "FaultMode" := TRUE;
   ELSE
       "FaultMode" := FALSE;
   END_IF;
END_FUNCTION_BLOCK

FUNCTION_BLOCK "MODES_STL"   // FB17, STL
{ S7_Optimized_Access := 'TRUE' }
VERSION : 0.1
   VAR
      OS1 : Bool;
      OS2 : Bool;
      OS3 : Bool;
      OS4 : Bool;
      OS5 : Bool;
   END_VAR
   VAR_TEMP
      TV1 : Time;
      T1 : Time;
      WMT : Bool;
      TV2 : Time;
      SMT : Bool;
      T2 : Time;
      StabilizekW_Min : Int;
      StabilizekW_Max : Int;
      TV3 : Time;
      T3 : Time;
      CMT : Bool;
   END_VAR
BEGIN

REGION Network 1: Warmup Mode
   // When Start pushbutton is pressed, the sequence begins with this step. Allow the rotor to turn at a speed somewhere between 20 and 50 RPMs and run the oil pump at some low output level (2- 10 GPM maybe?) until the oil temp reaches 150 degrees. Once we’ve maintained at least 150 degrees for 10 seconds, we want to transition into the next mode.
   EStopOrBrakeFailureAlarm:A     "EStopAlarm";
         O     "BrakeFailureAlarm";
         JC    SetAllAlarmTransitions;
         JU    RotorOverspeedOrHighOilTempAlarm;

   SetAllAlarmTransitions:S     "WarmupTransition";
         S     "StabilizeTransition";
         S     "GenerationTransition";
         S     "CooldownTransition";
         JU    StartSequenceBitCheck;

   RotorOverspeedOrHighOilTempAlarm:A     "RotorOverspeedAlarm";
         O     "HighOilTempAlarm";
         JC    SetSomeAlarmTransitions;
         JU    StartSequenceBitCheck;

   SetSomeAlarmTransitions:S     "WarmupTransition";
         S     "StabilizeTransition";
         S     "GenerationTransition";
         JU    StartSequenceBitCheck;

   StartSequenceBitCheck:A     "SystemStart_PB";
         A     "IdleMode";
         A     "FullAutoBit";
         FP    #OS1;
         JC    SetStartSequenceBit;
         JU    ResetStartSequenceBit;

   SetStartSequenceBit:S     "StartSequenceBit";
         JU    WarmupModeCheck;

   ResetStartSequenceBit:R     "StartSequenceBit";
         JU    WarmupModeCheck;

   WarmupModeCheck:A     "WarmupMode";
         JC    WarmupMode;
         JU    ResetWarmupModeTransition;

   WarmupMode:L     "WarmupRPM";
         T     "BafflePID_SP";
         L     "RPM";
         T     "BafflePID_In";
         S     "Baffle_Ctrl";
         S     "OilPumpVFD_Ctrl";
         R     "Brake_Ctrl";
         L     "WarmupVFD_Pct";
         T     "VFD_SP";
         L     "OilTemp";
         L     "WarmupOilTemp_SP";
         >=I;
         JC    WarmupModeTimer;
         JU    WarmupModeTimerReset;

   WarmupModeTimer:CALL  "MOVE"
         ( Int1  := "WarmupOilTempDelay_SP",
           Time1 := #TV1
         );
         CALL  TON, "IEC_Timer_0_DB_35"
         ( IN := TRUE,
           PT := #TV1,
           Q  := #WMT,
           ET := #T1
         );
         JU    WarmupModeTransitionCheck;

   WarmupModeTimerReset:CALL  RESET_TIMER
         ( "TIMER" := "IEC_Timer_0_DB_35"
         );
         JU    WarmupModeTransitionCheck;

   WarmupModeTransitionCheck:SET;
         A     #WMT;
         FP    #OS2;
         JC    SetWarmupModeTransition;
         JU    StabilizeModeCheck;

   SetWarmupModeTransition:CALL  RESET_TIMER
         ( "TIMER" := "IEC_Timer_0_DB_35"
         );
         SET;
         S     "WarmupTransition";
         JU    StabilizeModeCheck;

   ResetWarmupModeTransition:R     "WarmupTransition";
         JU    StabilizeModeCheck;
END_REGION

REGION Network 2: Stabilize Mode
   // Generator should speed up until desired kW output is attained. Once we’re stable within 5kW (+/-) of the setpoint for at least 10 seconds, we should transition into the next mode.
   StabilizeModeCheck:SET;
         A     "StabilizeMode";
         JC    StabilizeMode;
         JU    ResetStabilizeModeTransition;

   StabilizeMode:L     "Current";
         T     "BafflePID_In";
         L     "StabilizekW_SP";
         T     "BafflePID_SP";
         S     "Baffle_Ctrl";
         L     "StabilizekW_SP";
         L     5;
         -I;
         T     #StabilizekW_Min;
         L     "StabilizekW_SP";
         L     5;
         +I;
         T     #StabilizekW_Max;
         L     "Current";
         L     #StabilizekW_Min;
         <I;
         JC    StabilizeModeTimerReset;
         L     "Current";
         L     #StabilizekW_Max;
         >I;
         JC    StabilizeModeTimerReset;
         JU    StabilizeModeTimer;

   StabilizeModeTimerReset:CALL  RESET_TIMER
         ( "TIMER" := "IEC_Timer_0_DB_36"
         );
         JU    StabilizeModeTransitionCheck;

   StabilizeModeTimer:CALL  "MOVE"
         ( Int1  := "StabilizeDelay_SP",
           Time1 := #TV2
         );
         CALL  TON, "IEC_Timer_0_DB_36"
         ( IN := TRUE,
           PT := #TV2,
           Q  := #SMT,
           ET := #T2
         );
         JU    StabilizeModeTransitionCheck;

   StabilizeModeTransitionCheck:SET;
         A     #SMT;
         FP    #OS3;
         JC    SetStabilizeModeTransition;
         JU    GenerationModeCheck;

   SetStabilizeModeTransition:CALL  RESET_TIMER
         ( "TIMER" := "IEC_Timer_0_DB_36"
         );
         SET;
         S     "StabilizeTransition";
         JU    GenerationModeCheck;

   ResetStabilizeModeTransition:R     "StabilizeTransition";
         JU    GenerationModeCheck;
END_REGION

REGION Network 3: Generation Mode
   // Keep everything running and close the interlock.
   GenerationModeCheck:SET;
         A     "GenerationMode";
         JC    GenerationMode;
         JU    ResetGenerationModeTransition;

   GenerationMode:S     "StationInt_Ctrl";
         A     "SystemStop_PB";
         FP    #OS4;
         JC    SetGenerationModeTransition;
         O     "OvercurrentAlarm";
         JC    SetGenerationModeTransition;
         JU    ResetGenerationModeTransition;

   SetGenerationModeTransition:S     "GenerationTransition";
         JU    CooldownModeCheck;

   ResetGenerationModeTransition:R     "GenerationTransition";
         JU    CooldownModeCheck;
END_REGION

REGION Network 4: Cooldown Mode
   // Once the Stop button has been pushed, open the interlock, slow the rotor to between 20 and 50 RPMs and maintain a high oil flow until the oil temp is below 150 degrees. Once we’re below for ten seconds, we transition into Idle mode.
   CooldownModeCheck:SET;
         A     "CooldownMode";
         JC    CooldownMode;
         JU    ResetCooldownModeTransition;

   CooldownMode:R     "StationInt_Ctrl";
         L     "CooldownRPM";
         T     "BafflePID_SP";
         L     "RPM";
         T     "BafflePID_In";
         L     "OilTemp";
         L     "CooldownOilTemp_SP";
         <=I;
         JC    CooldownModeTimer;
         JU    CooldownModeTimerReset;

   CooldownModeTimer:CALL  "MOVE"
         ( Int1  := "CooldownDelay_SP",
           Time1 := #TV3
         );
         CALL  TON, "IEC_Timer_0_DB_37"
         ( IN := TRUE,
           PT := #TV3,
           Q  := #CMT,
           ET := #T3
         );
         JU    CooldownModeTransitionCheck;

   CooldownModeTimerReset:CALL  RESET_TIMER
         ( "TIMER" := "IEC_Timer_0_DB_37"
         );
         JU    CooldownModeTransitionCheck;

   CooldownModeTransitionCheck:SET;
         A     #CMT;
         FP    #OS5;
         JC    SetCooldownModeTransition;
         JU    IdleModeCheck;

   SetCooldownModeTransition:CALL  RESET_TIMER
         ( "TIMER" := "IEC_Timer_0_DB_37"
         );
         SET;
         S     "CooldownTransition";
         JU    IdleModeCheck;

   ResetCooldownModeTransition:R     "CooldownTransition";
         JU    IdleModeCheck;
END_REGION

REGION Network 5: Idle Mode
   // Interlock and baffle are deenergized and brake is engaged.
   IdleModeCheck:SET;
         A     "IdleMode";
         JC    IdleMode;
         JU    FaultModeCheck;

   IdleMode:R     "StationInt_Ctrl";
         R     "Baffle_Ctrl";
         R     "OilPumpVFD_Ctrl";
         S     "Brake_Ctrl";
END_REGION

REGION Network 6: Fault Mode
   // When we hit an alarm, the sequence should be aborted according to the alarm details (above in the Alarms section), and we should go into Fault mode (which is not part of our sequence).
   FaultModeCheck:A     "OvercurrentAlarm";
         O     "HighOilTempAlarm";
         O     "RotorOverspeedAlarm";
         O     "OilLowFlowAlarm";
         O     "OilHighFlowAlarm";
         O     "EStopAlarm";
         O     "BrakeFailureAlarm";
         JC    FaultMode;
         R     "FaultMode";
         JU    EndOfLine;

   FaultMode:S     "FaultMode";
         JU    EndOfLine;

   EndOfLine:BE;
END_REGION
END_FUNCTION_BLOCK

